LIN {X 0,Y 420.936,Z 312.19,A -85,B 0,C 180,E1 -10145.593,E2 -10145.593} C_VEL
LIN {X 0,Y 420.608,Z 319.802,A -85,B 0,C 180,E1 -10147.066,E2 -10147.066} C_VEL
LIN {X 0,Y 419.67,Z 336.36,A -85,B 0,C 180,E1 -10150.229,E2 -10150.229} C_VEL
LIN {X 0,Y 419.347,Z 341.705,A -85,B 0,C 180,E1 -10151.243,E2 -10151.243} C_VEL
LIN {X 0,Y 423.117,Z 368.844,A -85,B 0,C 180,E1 -10151.869,E2 -10151.869} C_VEL
LIN {X 0,Y 422.215,Z 450.861,A -85,B 0,C 180,E1 -10153.283,E2 -10153.283} C_VEL
LIN {X 0,Y 421.716,Z 464.725,A -85,B 0,C 180,E1 -10153.73,E2 -10153.73} C_VEL
LIN {X 0,Y 421.153,Z 477.157,A -85,B 0,C 180,E1 -10154.329,E2 -10154.329} C_VEL
LIN {X 0,Y 420.469,Z 489.063,A -85,B 0,C 180,E1 -10155.109,E2 -10155.109} C_VEL
LIN {X 0,Y 419.724,Z 501.027,A -85,B 0,C 180,E1 -10156.121,E2 -10156.121} C_VEL
LIN {X 0,Y 419.11,Z 510.84,A -85,B 0,C 180,E1 -10157.163,E2 -10157.163} C_VEL
LIN {X 0,Y 418.517,Z 520.102,A -85,B 0,C 180,E1 -10158.375,E2 -10158.375} C_VEL
LIN {X 0,Y 417.911,Z 529.108,A -85,B 0,C 180,E1 -10159.83,E2 -10159.83} C_VEL
LIN {X 0,Y 417.535,Z 536.352,A -85,B 0,C 180,E1 -10161.287,E2 -10161.287} C_VEL
LIN {X 0,Y 417.265,Z 542.12,A -85,B 0,C 180,E1 -10162.743,E2 -10162.743} C_VEL
LIN {X 0,Y 417.096,Z 546.655,A -85,B 0,C 180,E1 -10164.198,E2 -10164.198} C_VEL
LIN {X 0,Y 417.128,Z 549.047,A -85,B 0,C 180,E1 -10165.168,E2 -10165.168} C_VEL
LIN {X 0,Y 417.017,Z 550.997,A -85,B 0,C 180,E1 -10166.135,E2 -10166.135} C_VEL
LIN {X 0,Y 417.061,Z 552.532,A -85,B 0,C 180,E1 -10167.103,E2 -10167.103} C_VEL
LIN {X 0,Y 417.072,Z 553.609,A -85,B 0,C 180,E1 -10168.069,E2 -10168.069} C_VEL
LIN {X 0,Y 417.027,Z 554.572,A -85,B 0,C 180,E1 -10170.001,E2 -10170.001} C_VEL
LIN {X 0,Y 417.013,Z 554.471,A -85,B 0,C 180,E1 -10170.966,E2 -10170.966} C_VEL
LIN {X 0,Y 417.069,Z 553.941,A -85,B 0,C 180,E1 -10171.932,E2 -10171.932} C_VEL
LIN {X 0,Y 417.015,Z 551.682,A -85,B 0,C 180,E1 -10173.866,E2 -10173.866} C_VEL
LIN {X 0,Y 417.122,Z 548.885,A -85,B 0,C 180,E1 -10175.318,E2 -10175.318} C_VEL
LIN {X 0,Y 417.233,Z 545.071,A -85,B 0,C 180,E1 -10176.772,E2 -10176.772} C_VEL
LIN {X 0,Y 417.462,Z 540.144,A -85,B 0,C 180,E1 -10178.228,E2 -10178.228} C_VEL
LIN {X 0,Y 417.839,Z 533.958,A -85,B 0,C 180,E1 -10179.683,E2 -10179.683} C_VEL
LIN {X 0,Y 418.415,Z 526.279,A -85,B 0,C 180,E1 -10181.138,E2 -10181.138} C_VEL
LIN {X 0,Y 419.256,Z 516.655,A -85,B 0,C 180,E1 -10182.587,E2 -10182.587} C_VEL
LIN {X 0,Y 419.98,Z 506.28,A -85,B 0,C 180,E1 -10183.85,E2 -10183.85} C_VEL
LIN {X 0,Y 420.831,Z 495.628,A -85,B 0,C 180,E1 -10184.879,E2 -10184.879} C_VEL
LIN {X 0,Y 421.61,Z 484.753,A -85,B 0,C 180,E1 -10185.717,E2 -10185.717} C_VEL
LIN {X 0,Y 422.418,Z 472.754,A -85,B 0,C 180,E1 -10186.43,E2 -10186.43} C_VEL
LIN {X 0,Y 423.072,Z 459.606,A -85,B 0,C 180,E1 -10186.994,E2 -10186.994} C_VEL
LIN {X 0,Y 423.504,Z 446.445,A -85,B 0,C 180,E1 -10187.349,E2 -10187.349} C_VEL
LIN {X 0,Y 424.419,Z 367.986,A -85,B 0,C 180,E1 -10188.705,E2 -10188.705} C_VEL
LIN {X 0,Y 421.072,Z 347.455,A -85,B 0,C 180,E1 -10189.25,E2 -10189.25} C_VEL
LIN {X 0,Y 419.953,Z 341.257,A -85,B 0,C 180,E1 -10189.452,E2 -10189.452} C_VEL
LIN {X 0,Y 421.087,Z 324.061,A -85,B 0,C 180,E1 -10192.794,E2 -10192.794} C_VEL
LIN {X 0,Y 421.677,Z 314.787,A -85,B 0,C 180,E1 -10194.625,E2 -10194.625} C_VEL
LIN {X 0,Y 419.681,Z 304.414,A -85,B 0,C 180,E1 -10196.881,E2 -10196.881} C_VEL
LIN {X 0,Y 418.324,Z 298.383,A -85,B 0,C 180,E1 -10198.266,E2 -10198.266} C_VEL
LIN {X 0,Y 418.214,Z 298.393,A -85,B 0,C 180,E1 -10201.396,E2 -10201.396} C_VEL
LIN {X 0,Y 418.267,Z 298.386,A -85,B 0,C 180,E1 -10204.58,E2 -10204.58} C_VEL
LIN {X 0,Y 418.228,Z 298.389,A -85,B 0,C 180,E1 -10207.833,E2 -10207.833} C_VEL
LIN {X 0,Y 418.223,Z 298.389,A -85,B 0,C 180,E1 -10210.948,E2 -10210.948} C_VEL
LIN {X 0,Y 418.21,Z 298.389,A -85,B 0,C 180,E1 -10213.729,E2 -10213.729} C_VEL
LIN {X 0,Y 418.21,Z 298.393,A -85,B 0,C 180,E1 -10216.448,E2 -10216.448} C_VEL
LIN {X 0,Y 418.223,Z 298.386,A -85,B 0,C 180,E1 -10219.13,E2 -10219.13} C_VEL
LIN {X 0,Y 418.227,Z 298.386,A -85,B 0,C 180,E1 -10222.167,E2 -10222.167} C_VEL
LIN {X 0,Y 418.265,Z 298.378,A -85,B 0,C 180,E1 -10225.42,E2 -10225.42} C_VEL
LIN {X 0,Y 418.211,Z 298.39,A -85,B 0,C 180,E1 -10228.604,E2 -10228.604} C_VEL
LIN {X 0,Y 418.291,Z 298.377,A -85,B 0,C 180,E1 -10231.936,E2 -10231.936} C_VEL
LIN {X 0,Y 418.29,Z 298.383,A -85,B 0,C 180,E1 -10235.162,E2 -10235.162} C_VEL
LIN {X 0,Y 418.233,Z 298.383,A -85,B 0,C 180,E1 -10238.303,E2 -10238.303} C_VEL
LIN {X 0,Y 418.283,Z 298.379,A -85,B 0,C 180,E1 -10241.383,E2 -10241.383} C_VEL
LIN {X 0,Y 418.302,Z 298.373,A -85,B 0,C 180,E1 -10244.406,E2 -10244.406} C_VEL
LIN {X 0,Y 418.354,Z 298.37,A -85,B 0,C 180,E1 -10247.385,E2 -10247.385} C_VEL
LIN {X 0,Y 418.34,Z 298.367,A -85,B 0,C 180,E1 -10250.328,E2 -10250.328} C_VEL
LIN {X 0,Y 418.491,Z 298.351,A -85,B 0,C 180,E1 -10253.249,E2 -10253.249} C_VEL
LIN {X 0,Y 418.338,Z 298.365,A -85,B 0,C 180,E1 -10255.181,E2 -10255.181} C_VEL
LIN {X 0,Y 418.541,Z 298.343,A -85,B 0,C 180,E1 -10258.075,E2 -10258.075} C_VEL
LIN {X 0,Y 418.669,Z 298.329,A -85,B 0,C 180,E1 -10260,E2 -10260} C_VEL
LIN {X 0,Y 418.5,Z 298.344,A -85,B 0,C 180,E1 -10262.888,E2 -10262.888} C_VEL
LIN {X 0,Y 418.489,Z 298.349,A -85,B 0,C 180,E1 -10266.751,E2 -10266.751} C_VEL
LIN {X 0,Y 418.399,Z 298.364,A -85,B 0,C 180,E1 -10268.695,E2 -10268.695} C_VEL
LIN {X 0,Y 418.313,Z 298.372,A -85,B 0,C 180,E1 -10271.631,E2 -10271.631} C_VEL
LIN {X 0,Y 418.302,Z 298.381,A -85,B 0,C 180,E1 -10274.597,E2 -10274.597} C_VEL
LIN {X 0,Y 418.287,Z 298.376,A -85,B 0,C 180,E1 -10277.604,E2 -10277.604} C_VEL
LIN {X 0,Y 418.249,Z 298.384,A -85,B 0,C 180,E1 -10280.663,E2 -10280.663} C_VEL
LIN {X 0,Y 418.276,Z 298.377,A -85,B 0,C 180,E1 -10283.782,E2 -10283.782} C_VEL
LIN {X 0,Y 418.309,Z 298.376,A -85,B 0,C 180,E1 -10287.07,E2 -10287.07} C_VEL
LIN {X 0,Y 418.243,Z 298.382,A -85,B 0,C 180,E1 -10290.272,E2 -10290.272} C_VEL
LIN {X 0,Y 418.247,Z 298.382,A -85,B 0,C 180,E1 -10293.677,E2 -10293.677} C_VEL
LIN {X 0,Y 418.239,Z 298.386,A -85,B 0,C 180,E1 -10297.224,E2 -10297.224} C_VEL
LIN {X 0,Y 418.246,Z 298.383,A -85,B 0,C 180,E1 -10299.683,E2 -10299.683} C_VEL
LIN {X 0,Y 418.229,Z 298.385,A -85,B 0,C 180,E1 -10302.321,E2 -10302.321} C_VEL
LIN {X 0,Y 418.235,Z 298.387,A -85,B 0,C 180,E1 -10305.109,E2 -10305.109} C_VEL
LIN {X 0,Y 418.239,Z 298.388,A -85,B 0,C 180,E1 -10307.767,E2 -10307.767} C_VEL
LIN {X 0,Y 418.245,Z 298.386,A -85,B 0,C 180,E1 -10310.621,E2 -10310.621} C_VEL
LIN {X 0,Y 418.243,Z 298.386,A -85,B 0,C 180,E1 -10313.976,E2 -10313.976} C_VEL
LIN {X 0,Y 418.242,Z 298.389,A -85,B 0,C 180,E1 -10317.302,E2 -10317.302} C_VEL
LIN {X 0,Y 420.231,Z 307.957,A -85,B 0,C 180,E1 -10319.608,E2 -10319.608} C_VEL
LIN {X 0,Y 420.352,Z 312.594,A -85,B 0,C 180,E1 -10320.628,E2 -10320.628} C_VEL
LIN {X 0,Y 424.73,Z 331.843,A -85,B 0,C 180,E1 -10321.226,E2 -10321.226} C_VEL
LIN {X 0,Y 424.235,Z 375.558,A -85,B 0,C 180,E1 -10321.98,E2 -10321.98} C_VEL
LIN {X 0,Y 423.578,Z 420.934,A -85,B 0,C 180,E1 -10322.786,E2 -10322.786} C_VEL
LIN {X 0,Y 423.113,Z 434.256,A -85,B 0,C 180,E1 -10323.221,E2 -10323.221} C_VEL
LIN {X 0,Y 422.72,Z 446.148,A -85,B 0,C 180,E1 -10323.801,E2 -10323.801} C_VEL
LIN {X 0,Y 422.119,Z 456.766,A -85,B 0,C 180,E1 -10324.481,E2 -10324.481} C_VEL
LIN {X 0,Y 421.392,Z 467.515,A -85,B 0,C 180,E1 -10325.358,E2 -10325.358} C_VEL
LIN {X 0,Y 420.636,Z 477.399,A -85,B 0,C 180,E1 -10326.36,E2 -10326.36} C_VEL
LIN {X 0,Y 419.834,Z 487.413,A -85,B 0,C 180,E1 -10327.614,E2 -10327.614} C_VEL
LIN {X 0,Y 419.135,Z 495.554,A -85,B 0,C 180,E1 -10328.868,E2 -10328.868} C_VEL
LIN {X 0,Y 418.624,Z 502.01,A -85,B 0,C 180,E1 -10330.076,E2 -10330.076} C_VEL
LIN {X 0,Y 418.073,Z 507.767,A -85,B 0,C 180,E1 -10331.373,E2 -10331.373} C_VEL
LIN {X 0,Y 417.697,Z 513.126,A -85,B 0,C 180,E1 -10332.875,E2 -10332.875} C_VEL
LIN {X 0,Y 417.411,Z 517.248,A -85,B 0,C 180,E1 -10334.372,E2 -10334.372} C_VEL
LIN {X 0,Y 417.232,Z 519.362,A -85,B 0,C 180,E1 -10335.364,E2 -10335.364} C_VEL
LIN {X 0,Y 417.1,Z 521.024,A -85,B 0,C 180,E1 -10336.355,E2 -10336.355} C_VEL
LIN {X 0,Y 417.067,Z 522.941,A -85,B 0,C 180,E1 -10338.141,E2 -10338.141} C_VEL
LIN {X 0,Y 416.992,Z 523.472,A -85,B 0,C 180,E1 -10339.316,E2 -10339.316} C_VEL
LIN {X 0,Y 416.972,Z 523.075,A -85,B 0,C 180,E1 -10341.275,E2 -10341.275} C_VEL
LIN {X 0,Y 417.042,Z 522.162,A -85,B 0,C 180,E1 -10342.329,E2 -10342.329} C_VEL
LIN {X 0,Y 416.402,Z 521.209,A -85,B 0,C 180,E1 -10343.123,E2 -10343.123} C_VEL
LIN {X 0,Y 413.577,Z 519.17,A -85,B 0,C 180,E1 -10344.407,E2 -10344.407} C_VEL
LIN {X 0,Y 411.247,Z 517.028,A -85,B 0,C 180,E1 -10345.427,E2 -10345.427} C_VEL
LIN {X 0,Y 410.348,Z 515.063,A -85,B 0,C 180,E1 -10346.2,E2 -10346.2} C_VEL
LIN {X 0,Y 410.33,Z 514.318,A -85,B 0,C 180,E1 -10346.457,E2 -10346.457} C_VEL
LIN {X 0,Y 410.597,Z 509.016,A -85,B 0,C 180,E1 -10348.038,E2 -10348.038} C_VEL
LIN {X 0,Y 411.028,Z 502.734,A -85,B 0,C 180,E1 -10349.51,E2 -10349.51} C_VEL
LIN {X 0,Y 411.621,Z 494.875,A -85,B 0,C 180,E1 -10350.978,E2 -10350.978} C_VEL
LIN {X 0,Y 412.2,Z 485.137,A -85,B 0,C 180,E1 -10352.442,E2 -10352.442} C_VEL
LIN {X 0,Y 412.852,Z 474.969,A -85,B 0,C 180,E1 -10353.659,E2 -10353.659} C_VEL
LIN {X 0,Y 413.737,Z 464.843,A -85,B 0,C 180,E1 -10354.627,E2 -10354.627} C_VEL
LIN {X 0,Y 414.35,Z 453.869,A -85,B 0,C 180,E1 -10355.474,E2 -10355.474} C_VEL
LIN {X 0,Y 414.886,Z 441.713,A -85,B 0,C 180,E1 -10356.199,E2 -10356.199} C_VEL
LIN {X 0,Y 415.155,Z 428.961,A -85,B 0,C 180,E1 -10356.744,E2 -10356.744} C_VEL
LIN {X 0,Y 415.591,Z 416.702,A -85,B 0,C 180,E1 -10357.072,E2 -10357.072} C_VEL
LIN {X 0,Y 416.521,Z 332.666,A -85,B 0,C 180,E1 -10358.526,E2 -10358.526} C_VEL
LIN {X 0,Y 412.813,Z 312.758,A -85,B 0,C 180,E1 -10359.034,E2 -10359.034} C_VEL
LIN {X 0,Y 412.829,Z 308.131,A -85,B 0,C 180,E1 -10360.049,E2 -10360.049} C_VEL
LIN {X 0,Y 411.363,Z 299.247,A -85,B 0,C 180,E1 -10362.142,E2 -10362.142} C_VEL
LIN {X 0,Y 411.246,Z 299.256,A -85,B 0,C 180,E1 -10365.868,E2 -10365.868} C_VEL
LIN {X 0,Y 411.216,Z 299.259,A -85,B 0,C 180,E1 -10368.948,E2 -10368.948} C_VEL
LIN {X 0,Y 411.197,Z 299.266,A -85,B 0,C 180,E1 -10372.64,E2 -10372.64} C_VEL
LIN {X 0,Y 411.179,Z 299.263,A -85,B 0,C 180,E1 -10375.296,E2 -10375.296} C_VEL
LIN {X 0,Y 411.173,Z 299.27,A -85,B 0,C 180,E1 -10378.592,E2 -10378.592} C_VEL
LIN {X 0,Y 411.161,Z 299.265,A -85,B 0,C 180,E1 -10381.997,E2 -10381.997} C_VEL
LIN {X 0,Y 411.205,Z 299.266,A -85,B 0,C 180,E1 -10384.877,E2 -10384.877} C_VEL
LIN {X 0,Y 411.192,Z 299.261,A -85,B 0,C 180,E1 -10388.166,E2 -10388.166} C_VEL
LIN {X 0,Y 411.158,Z 299.265,A -85,B 0,C 180,E1 -10391.806,E2 -10391.806} C_VEL
LIN {X 0,Y 411.17,Z 299.266,A -85,B 0,C 180,E1 -10395.509,E2 -10395.509} C_VEL
LIN {X 0,Y 411.151,Z 299.268,A -85,B 0,C 180,E1 -10398.772,E2 -10398.772} C_VEL
LIN {X 0,Y 411.182,Z 299.262,A -85,B 0,C 180,E1 -10402.025,E2 -10402.025} C_VEL
LIN {X 0,Y 411.198,Z 299.264,A -85,B 0,C 180,E1 -10405.666,E2 -10405.666} C_VEL
LIN {X 0,Y 411.182,Z 299.265,A -85,B 0,C 180,E1 -10409.152,E2 -10409.152} C_VEL
LIN {X 0,Y 411.251,Z 299.253,A -85,B 0,C 180,E1 -10412.522,E2 -10412.522} C_VEL
LIN {X 0,Y 411.204,Z 299.265,A -85,B 0,C 180,E1 -10415.783,E2 -10415.783} C_VEL
LIN {X 0,Y 411.188,Z 299.261,A -85,B 0,C 180,E1 -10418.966,E2 -10418.966} C_VEL
LIN {X 0,Y 411.245,Z 299.258,A -85,B 0,C 180,E1 -10422.085,E2 -10422.085} C_VEL
LIN {X 0,Y 411.255,Z 299.253,A -85,B 0,C 180,E1 -10425.147,E2 -10425.147} C_VEL
LIN {X 0,Y 411.275,Z 299.256,A -85,B 0,C 180,E1 -10428.167,E2 -10428.167} C_VEL
LIN {X 0,Y 411.343,Z 299.242,A -85,B 0,C 180,E1 -10431.155,E2 -10431.155} C_VEL
LIN {X 0,Y 411.45,Z 299.236,A -85,B 0,C 180,E1 -10434.118,E2 -10434.118} C_VEL
LIN {X 0,Y 411.503,Z 299.227,A -85,B 0,C 180,E1 -10438.043,E2 -10438.043} C_VEL
LIN {X 0,Y 411.631,Z 299.21,A -85,B 0,C 180,E1 -10440,E2 -10440} C_VEL
LIN {X 0,Y 411.449,Z 299.23,A -85,B 0,C 180,E1 -10442.937,E2 -10442.937} C_VEL
LIN {X 0,Y 411.448,Z 299.232,A -85,B 0,C 180,E1 -10446.867,E2 -10446.867} C_VEL
LIN {X 0,Y 411.286,Z 299.249,A -85,B 0,C 180,E1 -10449.839,E2 -10449.839} C_VEL
LIN {X 0,Y 411.297,Z 299.25,A -85,B 0,C 180,E1 -10453.105,E2 -10453.105} C_VEL
LIN {X 0,Y 411.255,Z 299.259,A -85,B 0,C 180,E1 -10456.869,E2 -10456.869} C_VEL
LIN {X 0,Y 411.223,Z 299.257,A -85,B 0,C 180,E1 -10459.987,E2 -10459.987} C_VEL
LIN {X 0,Y 411.196,Z 299.265,A -85,B 0,C 180,E1 -10463.148,E2 -10463.148} C_VEL
LIN {X 0,Y 411.231,Z 299.257,A -85,B 0,C 180,E1 -10466.382,E2 -10466.382} C_VEL
LIN {X 0,Y 411.206,Z 299.26,A -85,B 0,C 180,E1 -10469.712,E2 -10469.712} C_VEL
LIN {X 0,Y 411.201,Z 299.267,A -85,B 0,C 180,E1 -10473.157,E2 -10473.157} C_VEL
LIN {X 0,Y 411.19,Z 299.261,A -85,B 0,C 180,E1 -10476.554,E2 -10476.554} C_VEL
LIN {X 0,Y 411.214,Z 299.261,A -85,B 0,C 180,E1 -10479.73,E2 -10479.73} C_VEL
LIN {X 0,Y 411.174,Z 299.266,A -85,B 0,C 180,E1 -10483.134,E2 -10483.134} C_VEL
LIN {X 0,Y 411.164,Z 299.267,A -85,B 0,C 180,E1 -10485.882,E2 -10485.882} C_VEL
LIN {X 0,Y 411.16,Z 299.265,A -85,B 0,C 180,E1 -10488.773,E2 -10488.773} C_VEL
LIN {X 0,Y 411.189,Z 299.265,A -85,B 0,C 180,E1 -10492.027,E2 -10492.027} C_VEL
LIN {X 0,Y 411.204,Z 299.265,A -85,B 0,C 180,E1 -10495.667,E2 -10495.667} C_VEL
LIN {X 0,Y 411.188,Z 299.261,A -85,B 0,C 180,E1 -10499.153,E2 -10499.153} C_VEL
LIN {X 0,Y 411.314,Z 299.353,A -85,B 0,C 180,E1 -10502.527,E2 -10502.527} C_VEL
LIN {X 0,Y 413.911,Z 312.994,A -85,B 0,C 180,E1 -10505.419,E2 -10505.419} C_VEL
LIN {X 0,Y 413.761,Z 319.175,A -85,B 0,C 180,E1 -10506.642,E2 -10506.642} C_VEL
LIN {X 0,Y 412.683,Z 336.91,A -85,B 0,C 180,E1 -10510.087,E2 -10510.087} C_VEL
LIN {X 0,Y 412.408,Z 341.367,A -85,B 0,C 180,E1 -10510.947,E2 -10510.947} C_VEL
LIN {X 0,Y 416.297,Z 369.883,A -85,B 0,C 180,E1 -10511.629,E2 -10511.629} C_VEL
LIN {X 0,Y 415.357,Z 450.171,A -85,B 0,C 180,E1 -10513.03,E2 -10513.03} C_VEL
LIN {X 0,Y 414.873,Z 463.413,A -85,B 0,C 180,E1 -10513.454,E2 -10513.454} C_VEL
LIN {X 0,Y 414.312,Z 476.161,A -85,B 0,C 180,E1 -10514.063,E2 -10514.063} C_VEL
LIN {X 0,Y 413.544,Z 488.258,A -85,B 0,C 180,E1 -10514.854,E2 -10514.854} C_VEL
LIN {X 0,Y 412.829,Z 499.823,A -85,B 0,C 180,E1 -10515.836,E2 -10515.836} C_VEL
LIN {X 0,Y 412.16,Z 510.297,A -85,B 0,C 180,E1 -10516.951,E2 -10516.951} C_VEL
LIN {X 0,Y 411.528,Z 519.568,A -85,B 0,C 180,E1 -10518.175,E2 -10518.175} C_VEL
LIN {X 0,Y 410.87,Z 528.62,A -85,B 0,C 180,E1 -10519.654,E2 -10519.654} C_VEL
LIN {X 0,Y 410.479,Z 535.909,A -85,B 0,C 180,E1 -10521.136,E2 -10521.136} C_VEL
LIN {X 0,Y 410.183,Z 541.721,A -85,B 0,C 180,E1 -10522.618,E2 -10522.618} C_VEL
LIN {X 0,Y 410.001,Z 546.289,A -85,B 0,C 180,E1 -10524.097,E2 -10524.097} C_VEL
LIN {X 0,Y 410.034,Z 548.697,A -85,B 0,C 180,E1 -10525.084,E2 -10525.084} C_VEL
LIN {X 0,Y 409.936,Z 550.662,A -85,B 0,C 180,E1 -10526.068,E2 -10526.068} C_VEL
LIN {X 0,Y 409.959,Z 552.214,A -85,B 0,C 180,E1 -10527.053,E2 -10527.053} C_VEL
LIN {X 0,Y 410,Z 553.313,A -85,B 0,C 180,E1 -10528.036,E2 -10528.036} C_VEL
LIN {X 0,Y 409.948,Z 554.301,A -85,B 0,C 180,E1 -10530.001,E2 -10530.001} C_VEL
LIN {X 0,Y 409.938,Z 554.216,A -85,B 0,C 180,E1 -10530.983,E2 -10530.983} C_VEL
LIN {X 0,Y 409.997,Z 553.708,A -85,B 0,C 180,E1 -10531.965,E2 -10531.965} C_VEL
LIN {X 0,Y 409.933,Z 551.474,A -85,B 0,C 180,E1 -10533.933,E2 -10533.933} C_VEL
LIN {X 0,Y 410.018,Z 548.704,A -85,B 0,C 180,E1 -10535.41,E2 -10535.41} C_VEL
LIN {X 0,Y 410.165,Z 544.919,A -85,B 0,C 180,E1 -10536.889,E2 -10536.889} C_VEL
LIN {X 0,Y 410.417,Z 540.024,A -85,B 0,C 180,E1 -10538.37,E2 -10538.37} C_VEL
LIN {X 0,Y 410.817,Z 533.875,A -85,B 0,C 180,E1 -10539.851,E2 -10539.851} C_VEL
LIN {X 0,Y 411.435,Z 526.251,A -85,B 0,C 180,E1 -10541.329,E2 -10541.329} C_VEL
LIN {X 0,Y 412.157,Z 518.468,A -85,B 0,C 180,E1 -10542.557,E2 -10542.557} C_VEL
LIN {X 0,Y 412.902,Z 508.984,A -85,B 0,C 180,E1 -10543.786,E2 -10543.786} C_VEL
LIN {X 0,Y 413.735,Z 498.496,A -85,B 0,C 180,E1 -10544.888,E2 -10544.888} C_VEL
LIN {X 0,Y 414.68,Z 486.836,A -85,B 0,C 180,E1 -10545.86,E2 -10545.86} C_VEL
LIN {X 0,Y 415.581,Z 474.397,A -85,B 0,C 180,E1 -10546.645,E2 -10546.645} C_VEL
LIN {X 0,Y 416.266,Z 461.319,A -85,B 0,C 180,E1 -10547.249,E2 -10547.249} C_VEL
LIN {X 0,Y 416.812,Z 448.275,A -85,B 0,C 180,E1 -10547.637,E2 -10547.637} C_VEL
LIN {X 0,Y 417.763,Z 368.347,A -85,B 0,C 180,E1 -10549.049,E2 -10549.049} C_VEL
LIN {X 0,Y 413.85,Z 345.109,A -85,B 0,C 180,E1 -10549.689,E2 -10549.689} C_VEL
LIN {X 0,Y 413.093,Z 341.048,A -85,B 0,C 180,E1 -10549.824,E2 -10549.824} C_VEL
LIN {X 0,Y 414.215,Z 325.143,A -85,B 0,C 180,E1 -10552.97,E2 -10552.97} C_VEL
LIN {X 0,Y 414.792,Z 317.366,A -85,B 0,C 180,E1 -10554.527,E2 -10554.527} C_VEL
LIN {X 0,Y 413.883,Z 311.29,A -85,B 0,C 180,E1 -10555.845,E2 -10555.845} C_VEL
LIN {X 0,Y 411.268,Z 299.263,A -85,B 0,C 180,E1 -10558.586,E2 -10558.586} C_VEL
LIN {X 0,Y 411.168,Z 299.273,A -85,B 0,C 180,E1 -10561.997,E2 -10561.997} C_VEL
LIN {X 0,Y 411.213,Z 299.262,A -85,B 0,C 180,E1 -10564.878,E2 -10564.878} C_VEL
LIN {X 0,Y 411.203,Z 299.265,A -85,B 0,C 180,E1 -10568.168,E2 -10568.168} C_VEL
LIN {X 0,Y 411.164,Z 299.267,A -85,B 0,C 180,E1 -10571.228,E2 -10571.228} C_VEL
LIN {X 0,Y 411.177,Z 299.268,A -85,B 0,C 180,E1 -10574.49,E2 -10574.49} C_VEL
LIN {X 0,Y 411.178,Z 299.265,A -85,B 0,C 180,E1 -10578.194,E2 -10578.194} C_VEL
LIN {X 0,Y 411.215,Z 299.263,A -85,B 0,C 180,E1 -10580.775,E2 -10580.775} C_VEL
LIN {X 0,Y 411.198,Z 299.263,A -85,B 0,C 180,E1 -10584.471,E2 -10584.471} C_VEL
LIN {X 0,Y 411.207,Z 299.261,A -85,B 0,C 180,E1 -10586.873,E2 -10586.873} C_VEL
LIN {X 0,Y 411.233,Z 299.256,A -85,B 0,C 180,E1 -10590.644,E2 -10590.644} C_VEL
LIN {X 0,Y 411.237,Z 299.257,A -85,B 0,C 180,E1 -10593.619,E2 -10593.619} C_VEL
LIN {X 0,Y 411.202,Z 299.262,A -85,B 0,C 180,E1 -10596.852,E2 -10596.852} C_VEL
LIN {X 0,Y 411.214,Z 299.258,A -85,B 0,C 180,E1 -10600.05,E2 -10600.05} C_VEL
LIN {X 0,Y 411.262,Z 299.254,A -85,B 0,C 180,E1 -10603.131,E2 -10603.131} C_VEL
LIN {X 0,Y 411.305,Z 299.244,A -85,B 0,C 180,E1 -10606.896,E2 -10606.896} C_VEL
LIN {X 0,Y 411.292,Z 299.246,A -85,B 0,C 180,E1 -10610.161,E2 -10610.161} C_VEL
LIN {X 0,Y 411.455,Z 299.226,A -85,B 0,C 180,E1 -10613.133,E2 -10613.133} C_VEL
LIN {X 0,Y 411.309,Z 299.24,A -85,B 0,C 180,E1 -10615.099,E2 -10615.099} C_VEL
LIN {X 0,Y 411.51,Z 299.219,A -85,B 0,C 180,E1 -10618.042,E2 -10618.042} C_VEL
LIN {X 0,Y 411.638,Z 299.204,A -85,B 0,C 180,E1 -10620,E2 -10620} C_VEL
LIN {X 0,Y 411.456,Z 299.221,A -85,B 0,C 180,E1 -10622.937,E2 -10622.937} C_VEL
LIN {X 0,Y 411.457,Z 299.224,A -85,B 0,C 180,E1 -10626.867,E2 -10626.867} C_VEL
LIN {X 0,Y 411.353,Z 299.241,A -85,B 0,C 180,E1 -10628.845,E2 -10628.845} C_VEL
LIN {X 0,Y 411.282,Z 299.249,A -85,B 0,C 180,E1 -10631.833,E2 -10631.833} C_VEL
LIN {X 0,Y 411.259,Z 299.255,A -85,B 0,C 180,E1 -10634.853,E2 -10634.853} C_VEL
LIN {X 0,Y 411.251,Z 299.254,A -85,B 0,C 180,E1 -10637.915,E2 -10637.915} C_VEL
LIN {X 0,Y 411.195,Z 299.263,A -85,B 0,C 180,E1 -10641.034,E2 -10641.034} C_VEL
LIN {X 0,Y 411.22,Z 299.258,A -85,B 0,C 180,E1 -10644.216,E2 -10644.216} C_VEL
LIN {X 0,Y 411.258,Z 299.25,A -85,B 0,C 180,E1 -10647.478,E2 -10647.478} C_VEL
LIN {X 0,Y 411.189,Z 299.265,A -85,B 0,C 180,E1 -10650.848,E2 -10650.848} C_VEL
LIN {X 0,Y 411.205,Z 299.258,A -85,B 0,C 180,E1 -10654.334,E2 -10654.334} C_VEL
LIN {X 0,Y 411.192,Z 299.261,A -85,B 0,C 180,E1 -10657.974,E2 -10657.974} C_VEL
LIN {X 0,Y 411.163,Z 299.27,A -85,B 0,C 180,E1 -10661.228,E2 -10661.228} C_VEL
LIN {X 0,Y 411.175,Z 299.264,A -85,B 0,C 180,E1 -10664.49,E2 -10664.49} C_VEL
LIN {X 0,Y 411.177,Z 299.265,A -85,B 0,C 180,E1 -10668.195,E2 -10668.195} C_VEL
LIN {X 0,Y 411.211,Z 299.262,A -85,B 0,C 180,E1 -10670.775,E2 -10670.775} C_VEL
LIN {X 0,Y 411.198,Z 299.261,A -85,B 0,C 180,E1 -10674.471,E2 -10674.471} C_VEL
LIN {X 0,Y 411.233,Z 299.389,A -85,B 0,C 180,E1 -10677.057,E2 -10677.057} C_VEL
LIN {X 0,Y 413.22,Z 308.79,A -85,B 0,C 180,E1 -10679.32,E2 -10679.32} C_VEL
LIN {X 0,Y 413.532,Z 312.859,A -85,B 0,C 180,E1 -10680.245,E2 -10680.245} C_VEL
LIN {X 0,Y 418.242,Z 333.489,A -85,B 0,C 180,E1 -10680.902,E2 -10680.902} C_VEL
LIN {X 0,Y 416.916,Z 420.997,A -85,B 0,C 180,E1 -10682.45,E2 -10682.45} C_VEL
LIN {X 0,Y 416.42,Z 434.381,A -85,B 0,C 180,E1 -10682.891,E2 -10682.891} C_VEL
LIN {X 0,Y 415.995,Z 446.833,A -85,B 0,C 180,E1 -10683.511,E2 -10683.511} C_VEL
LIN {X 0,Y 415.272,Z 458.615,A -85,B 0,C 180,E1 -10684.299,E2 -10684.299} C_VEL
LIN {X 0,Y 414.394,Z 470.373,A -85,B 0,C 180,E1 -10685.315,E2 -10685.315} C_VEL
LIN {X 0,Y 413.607,Z 480.137,A -85,B 0,C 180,E1 -10686.372,E2 -10686.372} C_VEL
LIN {X 0,Y 412.891,Z 488.541,A -85,B 0,C 180,E1 -10687.481,E2 -10687.481} C_VEL
LIN {X 0,Y 412.166,Z 496.511,A -85,B 0,C 180,E1 -10688.756,E2 -10688.756} C_VEL
LIN {X 0,Y 411.445,Z 504.231,A -85,B 0,C 180,E1 -10690.284,E2 -10690.284} C_VEL
LIN {X 0,Y 410.841,Z 511.303,A -85,B 0,C 180,E1 -10692.066,E2 -10692.066} C_VEL
LIN {X 0,Y 410.525,Z 515.604,A -85,B 0,C 180,E1 -10693.475,E2 -10693.475} C_VEL
LIN {X 0,Y 410.204,Z 519.386,A -85,B 0,C 180,E1 -10695.108,E2 -10695.108} C_VEL
LIN {X 0,Y 410.057,Z 521.094,A -85,B 0,C 180,E1 -10696.116,E2 -10696.116} C_VEL
LIN {X 0,Y 410.001,Z 522.933,A -85,B 0,C 180,E1 -10697.704,E2 -10697.704} C_VEL
LIN {X 0,Y 409.931,Z 523.716,A -85,B 0,C 180,E1 -10699.129,E2 -10699.129} C_VEL
LIN {X 0,Y 409.864,Z 523.406,A -85,B 0,C 180,E1 -10701.122,E2 -10701.122} C_VEL
LIN {X 0,Y 409.952,Z 522.397,A -85,B 0,C 180,E1 -10702.342,E2 -10702.342} C_VEL
LIN {X 0,Y 410.119,Z 519.889,A -85,B 0,C 180,E1 -10704.098,E2 -10704.098} C_VEL
LIN {X 0,Y 410.164,Z 516.71,A -85,B 0,C 180,E1 -10705.577,E2 -10705.577} C_VEL
LIN {X 0,Y 410.33,Z 514.318,A -85,B 0,C 180,E1 -10706.457,E2 -10706.457} C_VEL
LIN {X 0,Y 409.85,Z 512.038,A -85,B 0,C 180,E1 -10707.216,E2 -10707.216} C_VEL
LIN {X 0,Y 407.25,Z 507.932,A -85,B 0,C 180,E1 -10708.43,E2 -10708.43} C_VEL
LIN {X 0,Y 404.688,Z 503.127,A -85,B 0,C 180,E1 -10709.604,E2 -10709.604} C_VEL
LIN {X 0,Y 404.272,Z 499.747,A -85,B 0,C 180,E1 -10710.29,E2 -10710.29} C_VEL
LIN {X 0,Y 404.875,Z 491.372,A -85,B 0,C 180,E1 -10711.74,E2 -10711.74} C_VEL
LIN {X 0,Y 405.413,Z 482.595,A -85,B 0,C 180,E1 -10712.981,E2 -10712.981} C_VEL
LIN {X 0,Y 406.122,Z 472.94,A -85,B 0,C 180,E1 -10714.093,E2 -10714.093} C_VEL
LIN {X 0,Y 407.028,Z 462.319,A -85,B 0,C 180,E1 -10715.076,E2 -10715.076} C_VEL
LIN {X 0,Y 407.609,Z 450.524,A -85,B 0,C 180,E1 -10715.937,E2 -10715.937} C_VEL
LIN {X 0,Y 408.126,Z 438.264,A -85,B 0,C 180,E1 -10716.612,E2 -10716.612} C_VEL
LIN {X 0,Y 408.432,Z 426.605,A -85,B 0,C 180,E1 -10717.073,E2 -10717.073} C_VEL
LIN {X 0,Y 408.777,Z 414.179,A -85,B 0,C 180,E1 -10717.377,E2 -10717.377} C_VEL
LIN {X 0,Y 409.674,Z 333.501,A -85,B 0,C 180,E1 -10718.788,E2 -10718.788} C_VEL
LIN {X 0,Y 405.881,Z 312.872,A -85,B 0,C 180,E1 -10719.351,E2 -10719.351} C_VEL
LIN {X 0,Y 405.823,Z 308.965,A -85,B 0,C 180,E1 -10720.224,E2 -10720.224} C_VEL
LIN {X 0,Y 404.304,Z 300.126,A -85,B 0,C 180,E1 -10722.326,E2 -10722.326} C_VEL
LIN {X 0,Y 404.215,Z 300.135,A -85,B 0,C 180,E1 -10726.151,E2 -10726.151} C_VEL
LIN {X 0,Y 404.16,Z 300.137,A -85,B 0,C 180,E1 -10729.292,E2 -10729.292} C_VEL
LIN {X 0,Y 404.144,Z 300.142,A -85,B 0,C 180,E1 -10732.83,E2 -10732.83} C_VEL
LIN {X 0,Y 404.131,Z 300.14,A -85,B 0,C 180,E1 -10735.769,E2 -10735.769} C_VEL
LIN {X 0,Y 404.151,Z 300.138,A -85,B 0,C 180,E1 -10739.602,E2 -10739.602} C_VEL
LIN {X 0,Y 404.137,Z 300.145,A -85,B 0,C 180,E1 -10742.621,E2 -10742.621} C_VEL
LIN {X 0,Y 404.176,Z 300.138,A -85,B 0,C 180,E1 -10745.189,E2 -10745.189} C_VEL
LIN {X 0,Y 404.132,Z 300.145,A -85,B 0,C 180,E1 -10748.758,E2 -10748.758} C_VEL
LIN {X 0,Y 404.104,Z 300.145,A -85,B 0,C 180,E1 -10751.597,E2 -10751.597} C_VEL
LIN {X 0,Y 404.138,Z 300.141,A -85,B 0,C 180,E1 -10754.521,E2 -10754.521} C_VEL
LIN {X 0,Y 404.126,Z 300.147,A -85,B 0,C 180,E1 -10757.294,E2 -10757.294} C_VEL
LIN {X 0,Y 404.128,Z 300.141,A -85,B 0,C 180,E1 -10759.95,E2 -10759.95} C_VEL
LIN {X 0,Y 404.128,Z 300.145,A -85,B 0,C 180,E1 -10763.125,E2 -10763.125} C_VEL
LIN {X 0,Y 404.138,Z 300.14,A -85,B 0,C 180,E1 -10766.187,E2 -10766.187} C_VEL
LIN {X 0,Y 404.138,Z 300.144,A -85,B 0,C 180,E1 -10769.714,E2 -10769.714} C_VEL
LIN {X 0,Y 404.185,Z 300.135,A -85,B 0,C 180,E1 -10773.122,E2 -10773.122} C_VEL
LIN {X 0,Y 404.162,Z 300.14,A -85,B 0,C 180,E1 -10775.333,E2 -10775.333} C_VEL
LIN {X 0,Y 404.13,Z 300.14,A -85,B 0,C 180,E1 -10778.58,E2 -10778.58} C_VEL
LIN {X 0,Y 404.202,Z 300.138,A -85,B 0,C 180,E1 -10781.762,E2 -10781.762} C_VEL
LIN {X 0,Y 404.202,Z 300.131,A -85,B 0,C 180,E1 -10784.882,E2 -10784.882} C_VEL
LIN {X 0,Y 404.247,Z 300.133,A -85,B 0,C 180,E1 -10787.958,E2 -10787.958} C_VEL
LIN {X 0,Y 404.28,Z 300.121,A -85,B 0,C 180,E1 -10790.999,E2 -10790.999} C_VEL
LIN {X 0,Y 404.397,Z 300.113,A -85,B 0,C 180,E1 -10794.015,E2 -10794.015} C_VEL
LIN {X 0,Y 404.472,Z 300.102,A -85,B 0,C 180,E1 -10798.009,E2 -10798.009} C_VEL
LIN {X 0,Y 404.6,Z 300.085,A -85,B 0,C 180,E1 -10800,E2 -10800} C_VEL
LIN {X 0,Y 404.408,Z 300.107,A -85,B 0,C 180,E1 -10802.989,E2 -10802.989} C_VEL
LIN {X 0,Y 404.414,Z 300.107,A -85,B 0,C 180,E1 -10805.985,E2 -10805.985} C_VEL
LIN {X 0,Y 404.283,Z 300.123,A -85,B 0,C 180,E1 -10809.001,E2 -10809.001} C_VEL
LIN {X 0,Y 404.249,Z 300.127,A -85,B 0,C 180,E1 -10812.042,E2 -10812.042} C_VEL
LIN {X 0,Y 404.199,Z 300.134,A -85,B 0,C 180,E1 -10815.118,E2 -10815.118} C_VEL
LIN {X 0,Y 404.203,Z 300.133,A -85,B 0,C 180,E1 -10818.239,E2 -10818.239} C_VEL
LIN {X 0,Y 404.131,Z 300.142,A -85,B 0,C 180,E1 -10821.42,E2 -10821.42} C_VEL
LIN {X 0,Y 404.17,Z 300.139,A -85,B 0,C 180,E1 -10824.666,E2 -10824.666} C_VEL
LIN {X 0,Y 404.192,Z 300.132,A -85,B 0,C 180,E1 -10828,E2 -10828} C_VEL
LIN {X 0,Y 404.142,Z 300.142,A -85,B 0,C 180,E1 -10831.561,E2 -10831.561} C_VEL
LIN {X 0,Y 404.18,Z 300.139,A -85,B 0,C 180,E1 -10835.017,E2 -10835.017} C_VEL
LIN {X 0,Y 404.154,Z 300.138,A -85,B 0,C 180,E1 -10838.757,E2 -10838.757} C_VEL
LIN {X 0,Y 404.12,Z 300.147,A -85,B 0,C 180,E1 -10841.601,E2 -10841.601} C_VEL
LIN {X 0,Y 404.145,Z 300.138,A -85,B 0,C 180,E1 -10844.524,E2 -10844.524} C_VEL
LIN {X 0,Y 404.133,Z 300.144,A -85,B 0,C 180,E1 -10847.297,E2 -10847.297} C_VEL
LIN {X 0,Y 404.166,Z 300.14,A -85,B 0,C 180,E1 -10849.956,E2 -10849.956} C_VEL
LIN {X 0,Y 404.133,Z 300.141,A -85,B 0,C 180,E1 -10853.126,E2 -10853.126} C_VEL
LIN {X 0,Y 404.143,Z 300.142,A -85,B 0,C 180,E1 -10856.189,E2 -10856.189} C_VEL
LIN {X 0,Y 404.144,Z 300.144,A -85,B 0,C 180,E1 -10859.716,E2 -10859.716} C_VEL
LIN {X 0,Y 404.278,Z 300.228,A -85,B 0,C 180,E1 -10862.312,E2 -10862.312} C_VEL
LIN {X 0,Y 406.839,Z 313.779,A -85,B 0,C 180,E1 -10865.235,E2 -10865.235} C_VEL
LIN {X 0,Y 406.908,Z 318.838,A -85,B 0,C 180,E1 -10866.263,E2 -10866.263} C_VEL
LIN {X 0,Y 405.668,Z 337.712,A -85,B 0,C 180,E1 -10869.992,E2 -10869.992} C_VEL
LIN {X 0,Y 405.445,Z 341.182,A -85,B 0,C 180,E1 -10870.673,E2 -10870.673} C_VEL
LIN {X 0,Y 409.453,Z 369.811,A -85,B 0,C 180,E1 -10871.36,E2 -10871.36} C_VEL
LIN {X 0,Y 408.512,Z 449.408,A -85,B 0,C 180,E1 -10872.77,E2 -10872.77} C_VEL
LIN {X 0,Y 408.018,Z 462.826,A -85,B 0,C 180,E1 -10873.2,E2 -10873.2} C_VEL
LIN {X 0,Y 407.461,Z 475.092,A -85,B 0,C 180,E1 -10873.788,E2 -10873.788} C_VEL
LIN {X 0,Y 406.656,Z 487.432,A -85,B 0,C 180,E1 -10874.591,E2 -10874.591} C_VEL
LIN {X 0,Y 405.907,Z 499.098,A -85,B 0,C 180,E1 -10875.589,E2 -10875.589} C_VEL
LIN {X 0,Y 405.192,Z 509.867,A -85,B 0,C 180,E1 -10876.746,E2 -10876.746} C_VEL
LIN {X 0,Y 404.553,Z 519.022,A -85,B 0,C 180,E1 -10877.968,E2 -10877.968} C_VEL
LIN {X 0,Y 403.823,Z 528.119,A -85,B 0,C 180,E1 -10879.471,E2 -10879.471} C_VEL
LIN {X 0,Y 403.4,Z 535.451,A -85,B 0,C 180,E1 -10880.98,E2 -10880.98} C_VEL
LIN {X 0,Y 403.129,Z 541.313,A -85,B 0,C 180,E1 -10882.488,E2 -10882.488} C_VEL
LIN {X 0,Y 402.938,Z 545.916,A -85,B 0,C 180,E1 -10883.994,E2 -10883.994} C_VEL
LIN {X 0,Y 402.942,Z 548.343,A -85,B 0,C 180,E1 -10884.998,E2 -10884.998} C_VEL
LIN {X 0,Y 402.857,Z 550.323,A -85,B 0,C 180,E1 -10885.999,E2 -10885.999} C_VEL
LIN {X 0,Y 402.859,Z 551.889,A -85,B 0,C 180,E1 -10887.001,E2 -10887.001} C_VEL
LIN {X 0,Y 402.912,Z 553.016,A -85,B 0,C 180,E1 -10888.001,E2 -10888.001} C_VEL
LIN {X 0,Y 402.871,Z 554.031,A -85,B 0,C 180,E1 -10890.001,E2 -10890.001} C_VEL
LIN {X 0,Y 402.866,Z 553.958,A -85,B 0,C 180,E1 -10891,E2 -10891} C_VEL
LIN {X 0,Y 402.907,Z 553.476,A -85,B 0,C 180,E1 -10892,E2 -10892} C_VEL
LIN {X 0,Y 402.853,Z 551.269,A -85,B 0,C 180,E1 -10894.002,E2 -10894.002} C_VEL
LIN {X 0,Y 402.916,Z 548.527,A -85,B 0,C 180,E1 -10895.506,E2 -10895.506} C_VEL
LIN {X 0,Y 403.078,Z 544.773,A -85,B 0,C 180,E1 -10897.011,E2 -10897.011} C_VEL
LIN {X 0,Y 403.359,Z 539.912,A -85,B 0,C 180,E1 -10898.517,E2 -10898.517} C_VEL
LIN {X 0,Y 403.809,Z 533.801,A -85,B 0,C 180,E1 -10900.023,E2 -10900.023} C_VEL
LIN {X 0,Y 404.437,Z 526.225,A -85,B 0,C 180,E1 -10901.528,E2 -10901.528} C_VEL
LIN {X 0,Y 405.213,Z 518.501,A -85,B 0,C 180,E1 -10902.776,E2 -10902.776} C_VEL
LIN {X 0,Y 405.982,Z 509.1,A -85,B 0,C 180,E1 -10904.026,E2 -10904.026} C_VEL
LIN {X 0,Y 406.887,Z 498.69,A -85,B 0,C 180,E1 -10905.144,E2 -10905.144} C_VEL
LIN {X 0,Y 407.88,Z 487.147,A -85,B 0,C 180,E1 -10906.132,E2 -10906.132} C_VEL
LIN {X 0,Y 408.826,Z 474.947,A -85,B 0,C 180,E1 -10906.928,E2 -10906.928} C_VEL
LIN {X 0,Y 409.567,Z 461.403,A -85,B 0,C 180,E1 -10907.572,E2 -10907.572} C_VEL
LIN {X 0,Y 410.147,Z 448.686,A -85,B 0,C 180,E1 -10907.965,E2 -10907.965} C_VEL
LIN {X 0,Y 411.145,Z 369.032,A -85,B 0,C 180,E1 -10909.399,E2 -10909.399} C_VEL
LIN {X 0,Y 407.397,Z 346.781,A -85,B 0,C 180,E1 -10910.028,E2 -10910.028} C_VEL
LIN {X 0,Y 406.242,Z 340.683,A -85,B 0,C 180,E1 -10910.243,E2 -10910.243} C_VEL
LIN {X 0,Y 407.512,Z 324.026,A -85,B 0,C 180,E1 -10913.6,E2 -10913.6} C_VEL
LIN {X 0,Y 407.834,Z 317.361,A -85,B 0,C 180,E1 -10914.974,E2 -10914.974} C_VEL
LIN {X 0,Y 405.521,Z 305.678,A -85,B 0,C 180,E1 -10917.628,E2 -10917.628} C_VEL
LIN {X 0,Y 404.199,Z 300.142,A -85,B 0,C 180,E1 -10918.991,E2 -10918.991} C_VEL
LIN {X 0,Y 404.143,Z 300.141,A -85,B 0,C 180,E1 -10922.622,E2 -10922.622} C_VEL
LIN {X 0,Y 404.183,Z 300.137,A -85,B 0,C 180,E1 -10925.19,E2 -10925.19} C_VEL
LIN {X 0,Y 404.152,Z 300.144,A -85,B 0,C 180,E1 -10928.757,E2 -10928.757} C_VEL
LIN {X 0,Y 404.124,Z 300.144,A -85,B 0,C 180,E1 -10931.599,E2 -10931.599} C_VEL
LIN {X 0,Y 404.146,Z 300.143,A -85,B 0,C 180,E1 -10934.522,E2 -10934.522} C_VEL
LIN {X 0,Y 404.137,Z 300.141,A -85,B 0,C 180,E1 -10937.295,E2 -10937.295} C_VEL
LIN {X 0,Y 404.17,Z 300.134,A -85,B 0,C 180,E1 -10939.955,E2 -10939.955} C_VEL
LIN {X 0,Y 404.136,Z 300.142,A -85,B 0,C 180,E1 -10943.125,E2 -10943.125} C_VEL
LIN {X 0,Y 404.145,Z 300.136,A -85,B 0,C 180,E1 -10946.187,E2 -10946.187} C_VEL
LIN {X 0,Y 404.145,Z 300.138,A -85,B 0,C 180,E1 -10949.715,E2 -10949.715} C_VEL
LIN {X 0,Y 404.195,Z 300.134,A -85,B 0,C 180,E1 -10953.123,E2 -10953.123} C_VEL
LIN {X 0,Y 404.177,Z 300.141,A -85,B 0,C 180,E1 -10955.334,E2 -10955.334} C_VEL
LIN {X 0,Y 404.138,Z 300.139,A -85,B 0,C 180,E1 -10958.58,E2 -10958.58} C_VEL
LIN {X 0,Y 404.21,Z 300.132,A -85,B 0,C 180,E1 -10961.762,E2 -10961.762} C_VEL
LIN {X 0,Y 404.206,Z 300.13,A -85,B 0,C 180,E1 -10964.882,E2 -10964.882} C_VEL
LIN {X 0,Y 404.255,Z 300.126,A -85,B 0,C 180,E1 -10967.958,E2 -10967.958} C_VEL
LIN {X 0,Y 404.404,Z 300.107,A -85,B 0,C 180,E1 -10972.129,E2 -10972.129} C_VEL
LIN {X 0,Y 404.421,Z 300.101,A -85,B 0,C 180,E1 -10974.015,E2 -10974.015} C_VEL
LIN {X 0,Y 404.479,Z 300.095,A -85,B 0,C 180,E1 -10978.008,E2 -10978.008} C_VEL
LIN {X 0,Y 404.608,Z 300.08,A -85,B 0,C 180,E1 -10980,E2 -10980} C_VEL
LIN {X 0,Y 404.415,Z 300.098,A -85,B 0,C 180,E1 -10982.988,E2 -10982.988} C_VEL
LIN {X 0,Y 404.408,Z 300.102,A -85,B 0,C 180,E1 -10986.987,E2 -10986.987} C_VEL
LIN {X 0,Y 404.257,Z 300.127,A -85,B 0,C 180,E1 -10990.012,E2 -10990.012} C_VEL
LIN {X 0,Y 404.265,Z 300.123,A -85,B 0,C 180,E1 -10993.211,E2 -10993.211} C_VEL
LIN {X 0,Y 404.215,Z 300.132,A -85,B 0,C 180,E1 -10997.007,E2 -10997.007} C_VEL
LIN {X 0,Y 404.163,Z 300.139,A -85,B 0,C 180,E1 -11000.352,E2 -11000.352} C_VEL
LIN {X 0,Y 404.163,Z 300.136,A -85,B 0,C 180,E1 -11003.575,E2 -11003.575} C_VEL
LIN {X 0,Y 404.183,Z 300.133,A -85,B 0,C 180,E1 -11005.766,E2 -11005.766} C_VEL
LIN {X 0,Y 404.194,Z 300.129,A -85,B 0,C 180,E1 -11008,E2 -11008} C_VEL
LIN {X 0,Y 404.138,Z 300.138,A -85,B 0,C 180,E1 -11011.558,E2 -11011.558} C_VEL
LIN {X 0,Y 404.184,Z 300.135,A -85,B 0,C 180,E1 -11015.016,E2 -11015.016} C_VEL
LIN {X 0,Y 404.152,Z 300.14,A -85,B 0,C 180,E1 -11018.757,E2 -11018.757} C_VEL
LIN {X 0,Y 404.123,Z 300.146,A -85,B 0,C 180,E1 -11021.6,E2 -11021.6} C_VEL
LIN {X 0,Y 404.145,Z 300.14,A -85,B 0,C 180,E1 -11024.522,E2 -11024.522} C_VEL
LIN {X 0,Y 404.136,Z 300.145,A -85,B 0,C 180,E1 -11027.296,E2 -11027.296} C_VEL
LIN {X 0,Y 404.169,Z 300.14,A -85,B 0,C 180,E1 -11029.955,E2 -11029.955} C_VEL
LIN {X 0,Y 404.136,Z 300.144,A -85,B 0,C 180,E1 -11033.125,E2 -11033.125} C_VEL
LIN {X 0,Y 404.149,Z 300.145,A -85,B 0,C 180,E1 -11036.188,E2 -11036.188} C_VEL
LIN {X 0,Y 404.19,Z 300.255,A -85,B 0,C 180,E1 -11036.716,E2 -11036.716} C_VEL
LIN {X 0,Y 406.433,Z 310.922,A -85,B 0,C 180,E1 -11039.329,E2 -11039.329} C_VEL
LIN {X 0,Y 406.741,Z 313.458,A -85,B 0,C 180,E1 -11039.864,E2 -11039.864} C_VEL
LIN {X 0,Y 411.321,Z 332.813,A -85,B 0,C 180,E1 -11040.498,E2 -11040.498} C_VEL
LIN {X 0,Y 411.652,Z 336.493,A -85,B 0,C 180,E1 -11040.586,E2 -11040.586} C_VEL
LIN {X 0,Y 410.276,Z 421.133,A -85,B 0,C 180,E1 -11042.104,E2 -11042.104} C_VEL
LIN {X 0,Y 409.752,Z 434.476,A -85,B 0,C 180,E1 -11042.548,E2 -11042.548} C_VEL
LIN {X 0,Y 409.278,Z 447.158,A -85,B 0,C 180,E1 -11043.187,E2 -11043.187} C_VEL
LIN {X 0,Y 408.543,Z 458.826,A -85,B 0,C 180,E1 -11043.981,E2 -11043.981} C_VEL
LIN {X 0,Y 407.62,Z 470.59,A -85,B 0,C 180,E1 -11045.012,E2 -11045.012} C_VEL
LIN {X 0,Y 406.713,Z 481.267,A -85,B 0,C 180,E1 -11046.198,E2 -11046.198} C_VEL
LIN {X 0,Y 405.723,Z 491.292,A -85,B 0,C 180,E1 -11047.599,E2 -11047.599} C_VEL
LIN {X 0,Y 405.055,Z 498.828,A -85,B 0,C 180,E1 -11048.898,E2 -11048.898} C_VEL
LIN {X 0,Y 404.355,Z 506.177,A -85,B 0,C 180,E1 -11050.453,E2 -11050.453} C_VEL
LIN {X 0,Y 403.859,Z 511.09,A -85,B 0,C 180,E1 -11051.745,E2 -11051.745} C_VEL
LIN {X 0,Y 403.502,Z 515.904,A -85,B 0,C 180,E1 -11053.328,E2 -11053.328} C_VEL
LIN {X 0,Y 403.179,Z 519.387,A -85,B 0,C 180,E1 -11054.842,E2 -11054.842} C_VEL
LIN {X 0,Y 402.996,Z 521.167,A -85,B 0,C 180,E1 -11055.868,E2 -11055.868} C_VEL
LIN {X 0,Y 402.932,Z 523.201,A -85,B 0,C 180,E1 -11057.623,E2 -11057.623} C_VEL
LIN {X 0,Y 402.84,Z 523.958,A -85,B 0,C 180,E1 -11058.936,E2 -11058.936} C_VEL
LIN {X 0,Y 402.772,Z 523.736,A -85,B 0,C 180,E1 -11060.964,E2 -11060.964} C_VEL
LIN {X 0,Y 402.837,Z 523.04,A -85,B 0,C 180,E1 -11061.977,E2 -11061.977} C_VEL
LIN {X 0,Y 403.027,Z 520.895,A -85,B 0,C 180,E1 -11063.703,E2 -11063.703} C_VEL
LIN {X 0,Y 403.082,Z 517.3,A -85,B 0,C 180,E1 -11065.499,E2 -11065.499} C_VEL
LIN {X 0,Y 403.354,Z 513.15,A -85,B 0,C 180,E1 -11067.003,E2 -11067.003} C_VEL
LIN {X 0,Y 403.729,Z 506.839,A -85,B 0,C 180,E1 -11068.753,E2 -11068.753} C_VEL
LIN {X 0,Y 404.272,Z 499.747,A -85,B 0,C 180,E1 -11070.29,E2 -11070.29} C_VEL
LIN {X 0,Y 403.874,Z 496.243,A -85,B 0,C 180,E1 -11070.956,E2 -11070.956} C_VEL
LIN {X 0,Y 401.425,Z 490.177,A -85,B 0,C 180,E1 -11072.028,E2 -11072.028} C_VEL
LIN {X 0,Y 399.019,Z 483.664,A -85,B 0,C 180,E1 -11073.043,E2 -11073.043} C_VEL
LIN {X 0,Y 398.685,Z 479.284,A -85,B 0,C 180,E1 -11073.61,E2 -11073.61} C_VEL
LIN {X 0,Y 399.517,Z 468.24,A -85,B 0,C 180,E1 -11074.793,E2 -11074.793} C_VEL
LIN {X 0,Y 400.345,Z 457.955,A -85,B 0,C 180,E1 -11075.666,E2 -11075.666} C_VEL
LIN {X 0,Y 400.987,Z 445.727,A -85,B 0,C 180,E1 -11076.478,E2 -11076.478} C_VEL
LIN {X 0,Y 401.363,Z 432.203,A -85,B 0,C 180,E1 -11077.135,E2 -11077.135} C_VEL
LIN {X 0,Y 401.852,Z 419.076,A -85,B 0,C 180,E1 -11077.536,E2 -11077.536} C_VEL
LIN {X 0,Y 402.946,Z 334.691,A -85,B 0,C 180,E1 -11079.048,E2 -11079.048} C_VEL
LIN {X 0,Y 398.98,Z 313.15,A -85,B 0,C 180,E1 -11079.638,E2 -11079.638} C_VEL
LIN {X 0,Y 398.431,Z 307.579,A -85,B 0,C 180,E1 -11080.93,E2 -11080.93} C_VEL
LIN {X 0,Y 397.25,Z 301.005,A -85,B 0,C 180,E1 -11082.507,E2 -11082.507} C_VEL
LIN {X 0,Y 397.162,Z 301.015,A -85,B 0,C 180,E1 -11086.446,E2 -11086.446} C_VEL
LIN {X 0,Y 397.144,Z 301.011,A -85,B 0,C 180,E1 -11089.647,E2 -11089.647} C_VEL
LIN {X 0,Y 397.108,Z 301.017,A -85,B 0,C 180,E1 -11093.031,E2 -11093.031} C_VEL
LIN {X 0,Y 397.072,Z 301.023,A -85,B 0,C 180,E1 -11096.262,E2 -11096.262} C_VEL
LIN {X 0,Y 397.095,Z 301.017,A -85,B 0,C 180,E1 -11099.862,E2 -11099.862} C_VEL
LIN {X 0,Y 397.114,Z 301.014,A -85,B 0,C 180,E1 -11103.717,E2 -11103.717} C_VEL
LIN {X 0,Y 397.087,Z 301.021,A -85,B 0,C 180,E1 -11107.208,E2 -11107.208} C_VEL
LIN {X 0,Y 397.05,Z 301.024,A -85,B 0,C 180,E1 -11110.437,E2 -11110.437} C_VEL
LIN {X 0,Y 397.092,Z 301.018,A -85,B 0,C 180,E1 -11113.648,E2 -11113.648} C_VEL
LIN {X 0,Y 397.095,Z 301.018,A -85,B 0,C 180,E1 -11116.521,E2 -11116.521} C_VEL
LIN {X 0,Y 397.084,Z 301.018,A -85,B 0,C 180,E1 -11120.419,E2 -11120.419} C_VEL
LIN {X 0,Y 397.091,Z 301.021,A -85,B 0,C 180,E1 -11123.004,E2 -11123.004} C_VEL
LIN {X 0,Y 397.111,Z 301.015,A -85,B 0,C 180,E1 -11126.282,E2 -11126.282} C_VEL
LIN {X 0,Y 397.097,Z 301.017,A -85,B 0,C 180,E1 -11130.135,E2 -11130.135} C_VEL
LIN {X 0,Y 397.186,Z 301.005,A -85,B 0,C 180,E1 -11132.609,E2 -11132.609} C_VEL
LIN {X 0,Y 397.118,Z 301.018,A -85,B 0,C 180,E1 -11135.981,E2 -11135.981} C_VEL
LIN {X 0,Y 397.131,Z 301.019,A -85,B 0,C 180,E1 -11139.704,E2 -11139.704} C_VEL
LIN {X 0,Y 397.176,Z 301.006,A -85,B 0,C 180,E1 -11142.844,E2 -11142.844} C_VEL
LIN {X 0,Y 397.17,Z 301.011,A -85,B 0,C 180,E1 -11145.657,E2 -11145.657} C_VEL
LIN {X 0,Y 397.19,Z 301.005,A -85,B 0,C 180,E1 -11148.777,E2 -11148.777} C_VEL
LIN {X 0,Y 397.301,Z 300.998,A -85,B 0,C 180,E1 -11152.129,E2 -11152.129} C_VEL
LIN {X 0,Y 397.241,Z 300.999,A -85,B 0,C 180,E1 -11154.925,E2 -11154.925} C_VEL
LIN {X 0,Y 397.441,Z 300.977,A -85,B 0,C 180,E1 -11157.973,E2 -11157.973} C_VEL
LIN {X 0,Y 397.57,Z 300.961,A -85,B 0,C 180,E1 -11160,E2 -11160} C_VEL
LIN {X 0,Y 397.367,Z 300.984,A -85,B 0,C 180,E1 -11163.042,E2 -11163.042} C_VEL
LIN {X 0,Y 397.365,Z 300.986,A -85,B 0,C 180,E1 -11166.092,E2 -11166.092} C_VEL
LIN {X 0,Y 397.245,Z 300.999,A -85,B 0,C 180,E1 -11169.162,E2 -11169.162} C_VEL
LIN {X 0,Y 397.212,Z 301.005,A -85,B 0,C 180,E1 -11172.258,E2 -11172.258} C_VEL
LIN {X 0,Y 397.171,Z 301.008,A -85,B 0,C 180,E1 -11175.392,E2 -11175.392} C_VEL
LIN {X 0,Y 397.155,Z 301.014,A -85,B 0,C 180,E1 -11178.574,E2 -11178.574} C_VEL
LIN {X 0,Y 397.089,Z 301.017,A -85,B 0,C 180,E1 -11181.819,E2 -11181.819} C_VEL
LIN {X 0,Y 397.15,Z 301.015,A -85,B 0,C 180,E1 -11185.132,E2 -11185.132} C_VEL
LIN {X 0,Y 397.157,Z 301.009,A -85,B 0,C 180,E1 -11187.777,E2 -11187.777} C_VEL
LIN {X 0,Y 397.083,Z 301.022,A -85,B 0,C 180,E1 -11190.882,E2 -11190.882} C_VEL
LIN {X 0,Y 397.12,Z 301.014,A -85,B 0,C 180,E1 -11194.494,E2 -11194.494} C_VEL
LIN {X 0,Y 397.102,Z 301.016,A -85,B 0,C 180,E1 -11198.275,E2 -11198.275} C_VEL
LIN {X 0,Y 397.086,Z 301.02,A -85,B 0,C 180,E1 -11200.909,E2 -11200.909} C_VEL
LIN {X 0,Y 397.099,Z 301.021,A -85,B 0,C 180,E1 -11203.649,E2 -11203.649} C_VEL
LIN {X 0,Y 397.098,Z 301.016,A -85,B 0,C 180,E1 -11206.522,E2 -11206.522} C_VEL
LIN {X 0,Y 397.109,Z 301.015,A -85,B 0,C 180,E1 -11210.424,E2 -11210.424} C_VEL
LIN {X 0,Y 397.105,Z 301.017,A -85,B 0,C 180,E1 -11214.266,E2 -11214.266} C_VEL
LIN {X 0,Y 397.112,Z 301.014,A -85,B 0,C 180,E1 -11216.728,E2 -11216.728} C_VEL
LIN {X 0,Y 397.123,Z 301.018,A -85,B 0,C 180,E1 -11220.297,E2 -11220.297} C_VEL
LIN {X 0,Y 397.228,Z 301.152,A -85,B 0,C 180,E1 -11222.098,E2 -11222.098} C_VEL
LIN {X 0,Y 399.808,Z 314.566,A -85,B 0,C 180,E1 -11225.047,E2 -11225.047} C_VEL
LIN {X 0,Y 399.965,Z 319.268,A -85,B 0,C 180,E1 -11226.025,E2 -11226.025} C_VEL
LIN {X 0,Y 398.741,Z 337.192,A -85,B 0,C 180,E1 -11229.63,E2 -11229.63} C_VEL
LIN {X 0,Y 398.52,Z 340.954,A -85,B 0,C 180,E1 -11230.382,E2 -11230.382} C_VEL
LIN {X 0,Y 402.592,Z 369.998,A -85,B 0,C 180,E1 -11231.089,E2 -11231.089} C_VEL
LIN {X 0,Y 401.635,Z 449.749,A -85,B 0,C 180,E1 -11232.531,E2 -11232.531} C_VEL
LIN {X 0,Y 401.132,Z 462.965,A -85,B 0,C 180,E1 -11232.968,E2 -11232.968} C_VEL
LIN {X 0,Y 400.547,Z 475.129,A -85,B 0,C 180,E1 -11233.566,E2 -11233.566} C_VEL
LIN {X 0,Y 399.785,Z 486.578,A -85,B 0,C 180,E1 -11234.32,E2 -11234.32} C_VEL
LIN {X 0,Y 398.974,Z 498.358,A -85,B 0,C 180,E1 -11235.333,E2 -11235.333} C_VEL
LIN {X 0,Y 398.223,Z 509.468,A -85,B 0,C 180,E1 -11236.541,E2 -11236.541} C_VEL
LIN {X 0,Y 397.565,Z 518.458,A -85,B 0,C 180,E1 -11237.753,E2 -11237.753} C_VEL
LIN {X 0,Y 396.802,Z 527.609,A -85,B 0,C 180,E1 -11239.283,E2 -11239.283} C_VEL
LIN {X 0,Y 396.355,Z 534.986,A -85,B 0,C 180,E1 -11240.818,E2 -11240.818} C_VEL
LIN {X 0,Y 396.057,Z 540.892,A -85,B 0,C 180,E1 -11242.353,E2 -11242.353} C_VEL
LIN {X 0,Y 395.825,Z 546.317,A -85,B 0,C 180,E1 -11244.199,E2 -11244.199} C_VEL
LIN {X 0,Y 395.78,Z 549.981,A -85,B 0,C 180,E1 -11245.927,E2 -11245.927} C_VEL
LIN {X 0,Y 395.76,Z 551.561,A -85,B 0,C 180,E1 -11246.947,E2 -11246.947} C_VEL
LIN {X 0,Y 395.825,Z 552.717,A -85,B 0,C 180,E1 -11247.966,E2 -11247.966} C_VEL
LIN {X 0,Y 395.81,Z 553.432,A -85,B 0,C 180,E1 -11248.983,E2 -11248.983} C_VEL
LIN {X 0,Y 395.797,Z 553.76,A -85,B 0,C 180,E1 -11250.001,E2 -11250.001} C_VEL
LIN {X 0,Y 395.795,Z 553.701,A -85,B 0,C 180,E1 -11251.018,E2 -11251.018} C_VEL
LIN {X 0,Y 395.804,Z 553.244,A -85,B 0,C 180,E1 -11252.036,E2 -11252.036} C_VEL
LIN {X 0,Y 395.776,Z 551.067,A -85,B 0,C 180,E1 -11254.074,E2 -11254.074} C_VEL
LIN {X 0,Y 395.827,Z 547.932,A -85,B 0,C 180,E1 -11255.805,E2 -11255.805} C_VEL
LIN {X 0,Y 396.069,Z 543.176,A -85,B 0,C 180,E1 -11257.648,E2 -11257.648} C_VEL
LIN {X 0,Y 396.505,Z 536.938,A -85,B 0,C 180,E1 -11259.437,E2 -11259.437} C_VEL
LIN {X 0,Y 397.057,Z 530.169,A -85,B 0,C 180,E1 -11260.969,E2 -11260.969} C_VEL
LIN {X 0,Y 398.013,Z 521.786,A -85,B 0,C 180,E1 -11262.493,E2 -11262.493} C_VEL
LIN {X 0,Y 398.803,Z 513.17,A -85,B 0,C 180,E1 -11263.763,E2 -11263.763} C_VEL
LIN {X 0,Y 399.551,Z 504.108,A -85,B 0,C 180,E1 -11264.868,E2 -11264.868} C_VEL
LIN {X 0,Y 400.55,Z 493.521,A -85,B 0,C 180,E1 -11265.912,E2 -11265.912} C_VEL
LIN {X 0,Y 401.5,Z 482.343,A -85,B 0,C 180,E1 -11266.788,E2 -11266.788} C_VEL
LIN {X 0,Y 402.425,Z 469.815,A -85,B 0,C 180,E1 -11267.533,E2 -11267.533} C_VEL
LIN {X 0,Y 403.164,Z 456.441,A -85,B 0,C 180,E1 -11268.09,E2 -11268.09} C_VEL
LIN {X 0,Y 403.56,Z 444.093,A -85,B 0,C 180,E1 -11268.415,E2 -11268.415} C_VEL
LIN {X 0,Y 404.62,Z 370.41,A -85,B 0,C 180,E1 -11269.745,E2 -11269.745} C_VEL
LIN {X 0,Y 400.988,Z 348.632,A -85,B 0,C 180,E1 -11270.374,E2 -11270.374} C_VEL
LIN {X 0,Y 399.392,Z 340.4,A -85,B 0,C 180,E1 -11270.662,E2 -11270.662} C_VEL
LIN {X 0,Y 400.879,Z 322.836,A -85,B 0,C 180,E1 -11274.267,E2 -11274.267} C_VEL
LIN {X 0,Y 400.908,Z 318.657,A -85,B 0,C 180,E1 -11275.158,E2 -11275.158} C_VEL
LIN {X 0,Y 398.775,Z 307.818,A -85,B 0,C 180,E1 -11277.666,E2 -11277.666} C_VEL
LIN {X 0,Y 397.151,Z 301.021,A -85,B 0,C 180,E1 -11279.338,E2 -11279.338} C_VEL
LIN {X 0,Y 397.117,Z 301.015,A -85,B 0,C 180,E1 -11283.273,E2 -11283.273} C_VEL
LIN {X 0,Y 397.11,Z 301.02,A -85,B 0,C 180,E1 -11285.735,E2 -11285.735} C_VEL
LIN {X 0,Y 397.114,Z 301.018,A -85,B 0,C 180,E1 -11289.577,E2 -11289.577} C_VEL
LIN {X 0,Y 397.103,Z 301.018,A -85,B 0,C 180,E1 -11293.479,E2 -11293.479} C_VEL
LIN {X 0,Y 397.103,Z 301.021,A -85,B 0,C 180,E1 -11296.521,E2 -11296.521} C_VEL
LIN {X 0,Y 397.114,Z 301.015,A -85,B 0,C 180,E1 -11300.423,E2 -11300.423} C_VEL
LIN {X 0,Y 397.108,Z 301.016,A -85,B 0,C 180,E1 -11304.265,E2 -11304.265} C_VEL
LIN {X 0,Y 397.115,Z 301.015,A -85,B 0,C 180,E1 -11306.727,E2 -11306.727} C_VEL
LIN {X 0,Y 397.124,Z 301.012,A -85,B 0,C 180,E1 -11310.296,E2 -11310.296} C_VEL
LIN {X 0,Y 397.194,Z 301.006,A -85,B 0,C 180,E1 -11312.61,E2 -11312.61} C_VEL
LIN {X 0,Y 397.132,Z 301.012,A -85,B 0,C 180,E1 -11315.982,E2 -11315.982} C_VEL
LIN {X 0,Y 397.138,Z 301.014,A -85,B 0,C 180,E1 -11319.704,E2 -11319.704} C_VEL
LIN {X 0,Y 397.181,Z 301.006,A -85,B 0,C 180,E1 -11322.845,E2 -11322.845} C_VEL
LIN {X 0,Y 397.228,Z 300.997,A -85,B 0,C 180,E1 -11326.703,E2 -11326.703} C_VEL
LIN {X 0,Y 397.217,Z 300.999,A -85,B 0,C 180,E1 -11329.809,E2 -11329.809} C_VEL
LIN {X 0,Y 397.351,Z 300.982,A -85,B 0,C 180,E1 -11332.888,E2 -11332.888} C_VEL
LIN {X 0,Y 397.253,Z 300.99,A -85,B 0,C 180,E1 -11334.925,E2 -11334.925} C_VEL
LIN {X 0,Y 397.448,Z 300.971,A -85,B 0,C 180,E1 -11337.973,E2 -11337.973} C_VEL
LIN {X 0,Y 397.577,Z 300.955,A -85,B 0,C 180,E1 -11340,E2 -11340} C_VEL
LIN {X 0,Y 397.374,Z 300.975,A -85,B 0,C 180,E1 -11343.041,E2 -11343.041} C_VEL
LIN {X 0,Y 397.361,Z 300.979,A -85,B 0,C 180,E1 -11347.112,E2 -11347.112} C_VEL
LIN {X 0,Y 397.216,Z 301.006,A -85,B 0,C 180,E1 -11350.191,E2 -11350.191} C_VEL
LIN {X 0,Y 397.226,Z 300.999,A -85,B 0,C 180,E1 -11353.321,E2 -11353.321} C_VEL
LIN {X 0,Y 397.181,Z 301.007,A -85,B 0,C 180,E1 -11357.155,E2 -11357.155} C_VEL
LIN {X 0,Y 397.101,Z 301.017,A -85,B 0,C 180,E1 -11360.73,E2 -11360.73} C_VEL
LIN {X 0,Y 397.128,Z 301.012,A -85,B 0,C 180,E1 -11364.018,E2 -11364.018} C_VEL
LIN {X 0,Y 397.193,Z 301.003,A -85,B 0,C 180,E1 -11367.39,E2 -11367.39} C_VEL
LIN {X 0,Y 397.078,Z 301.021,A -85,B 0,C 180,E1 -11370.882,E2 -11370.882} C_VEL
LIN {X 0,Y 397.124,Z 301.013,A -85,B 0,C 180,E1 -11374.493,E2 -11374.493} C_VEL
LIN {X 0,Y 397.1,Z 301.016,A -85,B 0,C 180,E1 -11378.275,E2 -11378.275} C_VEL
LIN {X 0,Y 397.088,Z 301.019,A -85,B 0,C 180,E1 -11380.909,E2 -11380.909} C_VEL
LIN {X 0,Y 397.101,Z 301.022,A -85,B 0,C 180,E1 -11383.648,E2 -11383.648} C_VEL
LIN {X 0,Y 397.102,Z 301.018,A -85,B 0,C 180,E1 -11386.521,E2 -11386.521} C_VEL
LIN {X 0,Y 397.113,Z 301.019,A -85,B 0,C 180,E1 -11390.423,E2 -11390.423} C_VEL
LIN {X 0,Y 397.108,Z 301.017,A -85,B 0,C 180,E1 -11394.265,E2 -11394.265} C_VEL
LIN {X 0,Y 397.152,Z 301.186,A -85,B 0,C 180,E1 -11396.375,E2 -11396.375} C_VEL
LIN {X 0,Y 399.428,Z 311.776,A -85,B 0,C 180,E1 -11399.025,E2 -11399.025} C_VEL
LIN {X 0,Y 399.755,Z 313.697,A -85,B 0,C 180,E1 -11399.437,E2 -11399.437} C_VEL
LIN {X 0,Y 402.996,Z 325.761,A -85,B 0,C 180,E1 -11399.869,E2 -11399.869} C_VEL
LIN {X 0,Y 405.051,Z 335.285,A -85,B 0,C 180,E1 -11400.175,E2 -11400.175} C_VEL
LIN {X 0,Y 403.652,Z 421.352,A -85,B 0,C 180,E1 -11401.747,E2 -11401.747} C_VEL
LIN {X 0,Y 403.11,Z 435.192,A -85,B 0,C 180,E1 -11402.219,E2 -11402.219} C_VEL
LIN {X 0,Y 402.581,Z 447.93,A -85,B 0,C 180,E1 -11402.88,E2 -11402.88} C_VEL
LIN {X 0,Y 401.82,Z 459.061,A -85,B 0,C 180,E1 -11403.652,E2 -11403.652} C_VEL
LIN {X 0,Y 400.859,Z 470.825,A -85,B 0,C 180,E1 -11404.7,E2 -11404.7} C_VEL
LIN {X 0,Y 399.912,Z 481.547,A -85,B 0,C 180,E1 -11405.911,E2 -11405.911} C_VEL
LIN {X 0,Y 398.964,Z 490.703,A -85,B 0,C 180,E1 -11407.198,E2 -11407.198} C_VEL
LIN {X 0,Y 398.204,Z 498.379,A -85,B 0,C 180,E1 -11408.517,E2 -11408.517} C_VEL
LIN {X 0,Y 397.518,Z 505.05,A -85,B 0,C 180,E1 -11409.911,E2 -11409.911} C_VEL
LIN {X 0,Y 396.918,Z 510.878,A -85,B 0,C 180,E1 -11411.414,E2 -11411.414} C_VEL
LIN {X 0,Y 396.451,Z 516.251,A -85,B 0,C 180,E1 -11413.191,E2 -11413.191} C_VEL
LIN {X 0,Y 396.165,Z 519.372,A -85,B 0,C 180,E1 -11414.567,E2 -11414.567} C_VEL
LIN {X 0,Y 395.961,Z 521.239,A -85,B 0,C 180,E1 -11415.612,E2 -11415.612} C_VEL
LIN {X 0,Y 395.841,Z 523.483,A -85,B 0,C 180,E1 -11417.555,E2 -11417.555} C_VEL
LIN {X 0,Y 395.753,Z 524.172,A -85,B 0,C 180,E1 -11418.735,E2 -11418.735} C_VEL
LIN {X 0,Y 395.68,Z 524.331,A -85,B 0,C 180,E1 -11419.769,E2 -11419.769} C_VEL
LIN {X 0,Y 395.751,Z 523.41,A -85,B 0,C 180,E1 -11421.832,E2 -11421.832} C_VEL
LIN {X 0,Y 395.944,Z 521.165,A -85,B 0,C 180,E1 -11423.719,E2 -11423.719} C_VEL
LIN {X 0,Y 396.003,Z 517.884,A -85,B 0,C 180,E1 -11425.419,E2 -11425.419} C_VEL
LIN {X 0,Y 396.271,Z 513.83,A -85,B 0,C 180,E1 -11426.95,E2 -11426.95} C_VEL
LIN {X 0,Y 396.618,Z 507.625,A -85,B 0,C 180,E1 -11428.73,E2 -11428.73} C_VEL
LIN {X 0,Y 397.168,Z 500.868,A -85,B 0,C 180,E1 -11430.253,E2 -11430.253} C_VEL
LIN {X 0,Y 397.818,Z 492.469,A -85,B 0,C 180,E1 -11431.771,E2 -11431.771} C_VEL
LIN {X 0,Y 398.37,Z 483.855,A -85,B 0,C 180,E1 -11433.033,E2 -11433.033} C_VEL
LIN {X 0,Y 398.685,Z 479.284,A -85,B 0,C 180,E1 -11433.61,E2 -11433.61} C_VEL
LIN {X 0,Y 398.403,Z 474.779,A -85,B 0,C 180,E1 -11434.148,E2 -11434.148} C_VEL
LIN {X 0,Y 396.237,Z 467.198,A -85,B 0,C 180,E1 -11435.009,E2 -11435.009} C_VEL
LIN {X 0,Y 394.035,Z 459.169,A -85,B 0,C 180,E1 -11435.796,E2 -11435.796} C_VEL
LIN {X 0,Y 393.705,Z 453.903,A -85,B 0,C 180,E1 -11436.213,E2 -11436.213} C_VEL
LIN {X 0,Y 394.314,Z 441.435,A -85,B 0,C 180,E1 -11436.974,E2 -11436.974} C_VEL
LIN {X 0,Y 394.583,Z 429.097,A -85,B 0,C 180,E1 -11437.515,E2 -11437.515} C_VEL
LIN {X 0,Y 395.039,Z 417.893,A -85,B 0,C 180,E1 -11437.828,E2 -11437.828} C_VEL
LIN {X 0,Y 396.102,Z 335.419,A -85,B 0,C 180,E1 -11439.327,E2 -11439.327} C_VEL
LIN {X 0,Y 392.025,Z 313.463,A -85,B 0,C 180,E1 -11439.93,E2 -11439.93} C_VEL
LIN {X 0,Y 390.84,Z 305.081,A -85,B 0,C 180,E1 -11441.934,E2 -11441.934} C_VEL
LIN {X 0,Y 390.222,Z 301.88,A -85,B 0,C 180,E1 -11442.761,E2 -11442.761} C_VEL
LIN {X 0,Y 390.135,Z 301.886,A -85,B 0,C 180,E1 -11446.751,E2 -11446.751} C_VEL
LIN {X 0,Y 390.086,Z 301.897,A -85,B 0,C 180,E1 -11450.469,E2 -11450.469} C_VEL
LIN {X 0,Y 390.06,Z 301.893,A -85,B 0,C 180,E1 -11453.352,E2 -11453.352} C_VEL
LIN {X 0,Y 390.027,Z 301.903,A -85,B 0,C 180,E1 -11456.774,E2 -11456.774} C_VEL
LIN {X 0,Y 390.033,Z 301.899,A -85,B 0,C 180,E1 -11460.299,E2 -11460.299} C_VEL
LIN {X 0,Y 390.064,Z 301.893,A -85,B 0,C 180,E1 -11464.024,E2 -11464.024} C_VEL
LIN {X 0,Y 390.036,Z 301.897,A -85,B 0,C 180,E1 -11467.549,E2 -11467.549} C_VEL
LIN {X 0,Y 390.013,Z 301.904,A -85,B 0,C 180,E1 -11470.814,E2 -11470.814} C_VEL
LIN {X 0,Y 390.046,Z 301.895,A -85,B 0,C 180,E1 -11473.885,E2 -11473.885} C_VEL
LIN {X 0,Y 390.049,Z 301.897,A -85,B 0,C 180,E1 -11476.789,E2 -11476.789} C_VEL
LIN {X 0,Y 390.049,Z 301.898,A -85,B 0,C 180,E1 -11479.56,E2 -11479.56} C_VEL
LIN {X 0,Y 390.034,Z 301.896,A -85,B 0,C 180,E1 -11482.449,E2 -11482.449} C_VEL
LIN {X 0,Y 390.061,Z 301.894,A -85,B 0,C 180,E1 -11485.975,E2 -11485.975} C_VEL
LIN {X 0,Y 390.039,Z 301.899,A -85,B 0,C 180,E1 -11489.869,E2 -11489.869} C_VEL
LIN {X 0,Y 390.104,Z 301.891,A -85,B 0,C 180,E1 -11493.231,E2 -11493.231} C_VEL
LIN {X 0,Y 390.059,Z 301.893,A -85,B 0,C 180,E1 -11496.763,E2 -11496.763} C_VEL
LIN {X 0,Y 390.096,Z 301.893,A -85,B 0,C 180,E1 -11499.983,E2 -11499.983} C_VEL
LIN {X 0,Y 390.133,Z 301.885,A -85,B 0,C 180,E1 -11503.248,E2 -11503.248} C_VEL
LIN {X 0,Y 390.186,Z 301.878,A -85,B 0,C 180,E1 -11506.561,E2 -11506.561} C_VEL
LIN {X 0,Y 390.195,Z 301.877,A -85,B 0,C 180,E1 -11510.671,E2 -11510.671} C_VEL
LIN {X 0,Y 390.299,Z 301.866,A -85,B 0,C 180,E1 -11513.798,E2 -11513.798} C_VEL
LIN {X 0,Y 390.41,Z 301.853,A -85,B 0,C 180,E1 -11517.937,E2 -11517.937} C_VEL
LIN {X 0,Y 390.539,Z 301.837,A -85,B 0,C 180,E1 -11520,E2 -11520} C_VEL
LIN {X 0,Y 390.302,Z 301.863,A -85,B 0,C 180,E1 -11523.097,E2 -11523.097} C_VEL
LIN {X 0,Y 390.319,Z 301.865,A -85,B 0,C 180,E1 -11526.202,E2 -11526.202} C_VEL
LIN {X 0,Y 390.197,Z 301.876,A -85,B 0,C 180,E1 -11529.329,E2 -11529.329} C_VEL
LIN {X 0,Y 390.187,Z 301.878,A -85,B 0,C 180,E1 -11533.439,E2 -11533.439} C_VEL
LIN {X 0,Y 390.141,Z 301.885,A -85,B 0,C 180,E1 -11537.308,E2 -11537.308} C_VEL
LIN {X 0,Y 390.08,Z 301.893,A -85,B 0,C 180,E1 -11540.471,E2 -11540.471} C_VEL
LIN {X 0,Y 390.082,Z 301.893,A -85,B 0,C 180,E1 -11543.351,E2 -11543.351} C_VEL
LIN {X 0,Y 390.107,Z 301.891,A -85,B 0,C 180,E1 -11546.769,E2 -11546.769} C_VEL
LIN {X 0,Y 390.04,Z 301.896,A -85,B 0,C 180,E1 -11550.3,E2 -11550.3} C_VEL
LIN {X 0,Y 390.05,Z 301.896,A -85,B 0,C 180,E1 -11552.721,E2 -11552.721} C_VEL
LIN {X 0,Y 390.052,Z 301.896,A -85,B 0,C 180,E1 -11555.826,E2 -11555.826} C_VEL
LIN {X 0,Y 390.067,Z 301.898,A -85,B 0,C 180,E1 -11559.22,E2 -11559.22} C_VEL
LIN {X 0,Y 390.04,Z 301.895,A -85,B 0,C 180,E1 -11562.375,E2 -11562.375} C_VEL
LIN {X 0,Y 390.042,Z 301.901,A -85,B 0,C 180,E1 -11565.356,E2 -11565.356} C_VEL
LIN {X 0,Y 390.027,Z 301.898,A -85,B 0,C 180,E1 -11568.188,E2 -11568.188} C_VEL
LIN {X 0,Y 390.084,Z 301.89,A -85,B 0,C 180,E1 -11570.908,E2 -11570.908} C_VEL
LIN {X 0,Y 390.083,Z 301.89,A -85,B 0,C 180,E1 -11574.794,E2 -11574.794} C_VEL
LIN {X 0,Y 390.022,Z 301.899,A -85,B 0,C 180,E1 -11578.497,E2 -11578.497} C_VEL
LIN {X 0,Y 390.175,Z 301.97,A -85,B 0,C 180,E1 -11581.853,E2 -11581.853} C_VEL
LIN {X 0,Y 392.994,Z 316.705,A -85,B 0,C 180,E1 -11585.15,E2 -11585.15} C_VEL
LIN {X 0,Y 392.861,Z 322.058,A -85,B 0,C 180,E1 -11586.266,E2 -11586.266} C_VEL
LIN {X 0,Y 391.742,Z 337.982,A -85,B 0,C 180,E1 -11589.524,E2 -11589.524} C_VEL
LIN {X 0,Y 391.546,Z 340.626,A -85,B 0,C 180,E1 -11590.061,E2 -11590.061} C_VEL
LIN {X 0,Y 395.79,Z 371.41,A -85,B 0,C 180,E1 -11590.834,E2 -11590.834} C_VEL
LIN {X 0,Y 394.812,Z 448.867,A -85,B 0,C 180,E1 -11592.252,E2 -11592.252} C_VEL
LIN {X 0,Y 394.248,Z 462.289,A -85,B 0,C 180,E1 -11592.695,E2 -11592.695} C_VEL
LIN {X 0,Y 393.639,Z 475.138,A -85,B 0,C 180,E1 -11593.336,E2 -11593.336} C_VEL
LIN {X 0,Y 392.791,Z 487.311,A -85,B 0,C 180,E1 -11594.166,E2 -11594.166} C_VEL
LIN {X 0,Y 391.959,Z 498.902,A -85,B 0,C 180,E1 -11595.197,E2 -11595.197} C_VEL
LIN {X 0,Y 391.257,Z 509.048,A -85,B 0,C 180,E1 -11596.327,E2 -11596.327} C_VEL
LIN {X 0,Y 390.568,Z 517.872,A -85,B 0,C 180,E1 -11597.531,E2 -11597.531} C_VEL
LIN {X 0,Y 389.797,Z 527.091,A -85,B 0,C 180,E1 -11599.088,E2 -11599.088} C_VEL
LIN {X 0,Y 389.326,Z 534.515,A -85,B 0,C 180,E1 -11600.651,E2 -11600.651} C_VEL
LIN {X 0,Y 388.986,Z 540.46,A -85,B 0,C 180,E1 -11602.213,E2 -11602.213} C_VEL
LIN {X 0,Y 388.774,Z 545.362,A -85,B 0,C 180,E1 -11603.857,E2 -11603.857} C_VEL
LIN {X 0,Y 388.719,Z 548.697,A -85,B 0,C 180,E1 -11605.334,E2 -11605.334} C_VEL
LIN {X 0,Y 388.664,Z 551.231,A -85,B 0,C 180,E1 -11606.891,E2 -11606.891} C_VEL
LIN {X 0,Y 388.724,Z 552.412,A -85,B 0,C 180,E1 -11607.928,E2 -11607.928} C_VEL
LIN {X 0,Y 388.74,Z 553.147,A -85,B 0,C 180,E1 -11608.965,E2 -11608.965} C_VEL
LIN {X 0,Y 388.726,Z 553.488,A -85,B 0,C 180,E1 -11610.001,E2 -11610.001} C_VEL
LIN {X 0,Y 388.726,Z 553.444,A -85,B 0,C 180,E1 -11611.036,E2 -11611.036} C_VEL
LIN {X 0,Y 388.701,Z 553.008,A -85,B 0,C 180,E1 -11612.073,E2 -11612.073} C_VEL
LIN {X 0,Y 388.701,Z 550.868,A -85,B 0,C 180,E1 -11614.148,E2 -11614.148} C_VEL
LIN {X 0,Y 388.775,Z 547.28,A -85,B 0,C 180,E1 -11616.144,E2 -11616.144} C_VEL
LIN {X 0,Y 389.022,Z 543.055,A -85,B 0,C 180,E1 -11617.788,E2 -11617.788} C_VEL
LIN {X 0,Y 389.485,Z 536.86,A -85,B 0,C 180,E1 -11619.609,E2 -11619.609} C_VEL
LIN {X 0,Y 390.062,Z 530.133,A -85,B 0,C 180,E1 -11621.169,E2 -11621.169} C_VEL
LIN {X 0,Y 391.069,Z 521.815,A -85,B 0,C 180,E1 -11622.718,E2 -11622.718} C_VEL
LIN {X 0,Y 391.967,Z 512.088,A -85,B 0,C 180,E1 -11624.17,E2 -11624.17} C_VEL
LIN {X 0,Y 392.937,Z 501.726,A -85,B 0,C 180,E1 -11625.417,E2 -11625.417} C_VEL
LIN {X 0,Y 394.011,Z 490.967,A -85,B 0,C 180,E1 -11626.449,E2 -11626.449} C_VEL
LIN {X 0,Y 395.071,Z 479.064,A -85,B 0,C 180,E1 -11627.336,E2 -11627.336} C_VEL
LIN {X 0,Y 395.966,Z 466.703,A -85,B 0,C 180,E1 -11628.029,E2 -11628.029} C_VEL
LIN {X 0,Y 396.716,Z 453.959,A -85,B 0,C 180,E1 -11628.528,E2 -11628.528} C_VEL
LIN {X 0,Y 397.054,Z 440.112,A -85,B 0,C 180,E1 -11628.855,E2 -11628.855} C_VEL
LIN {X 0,Y 397.994,Z 370.779,A -85,B 0,C 180,E1 -11630.131,E2 -11630.131} C_VEL
LIN {X 0,Y 393.936,Z 347.003,A -85,B 0,C 180,E1 -11630.842,E2 -11630.842} C_VEL
LIN {X 0,Y 392.537,Z 340.2,A -85,B 0,C 180,E1 -11631.082,E2 -11631.082} C_VEL
LIN {X 0,Y 393.878,Z 325.133,A -85,B 0,C 180,E1 -11634.23,E2 -11634.23} C_VEL
LIN {X 0,Y 394.137,Z 321.08,A -85,B 0,C 180,E1 -11635.093,E2 -11635.093} C_VEL
LIN {X 0,Y 392.209,Z 310.918,A -85,B 0,C 180,E1 -11637.478,E2 -11637.478} C_VEL
LIN {X 0,Y 390.081,Z 301.902,A -85,B 0,C 180,E1 -11639.7,E2 -11639.7} C_VEL
LIN {X 0,Y 390.045,Z 301.896,A -85,B 0,C 180,E1 -11642.721,E2 -11642.721} C_VEL
LIN {X 0,Y 390.058,Z 301.899,A -85,B 0,C 180,E1 -11645.825,E2 -11645.825} C_VEL
LIN {X 0,Y 390.068,Z 301.895,A -85,B 0,C 180,E1 -11649.218,E2 -11649.218} C_VEL
LIN {X 0,Y 390.043,Z 301.9,A -85,B 0,C 180,E1 -11652.374,E2 -11652.374} C_VEL
LIN {X 0,Y 390.045,Z 301.898,A -85,B 0,C 180,E1 -11655.354,E2 -11655.354} C_VEL
LIN {X 0,Y 390.032,Z 301.899,A -85,B 0,C 180,E1 -11658.186,E2 -11658.186} C_VEL
LIN {X 0,Y 390.089,Z 301.895,A -85,B 0,C 180,E1 -11660.907,E2 -11660.907} C_VEL
LIN {X 0,Y 390.085,Z 301.896,A -85,B 0,C 180,E1 -11664.793,E2 -11664.793} C_VEL
LIN {X 0,Y 390.024,Z 301.9,A -85,B 0,C 180,E1 -11668.495,E2 -11668.495} C_VEL
LIN {X 0,Y 390.117,Z 301.886,A -85,B 0,C 180,E1 -11672.07,E2 -11672.07} C_VEL
LIN {X 0,Y 390.08,Z 301.895,A -85,B 0,C 180,E1 -11675.519,E2 -11675.519} C_VEL
LIN {X 0,Y 390.055,Z 301.896,A -85,B 0,C 180,E1 -11678.878,E2 -11678.878} C_VEL
LIN {X 0,Y 390.128,Z 301.884,A -85,B 0,C 180,E1 -11682.167,E2 -11682.167} C_VEL
LIN {X 0,Y 390.144,Z 301.882,A -85,B 0,C 180,E1 -11685.392,E2 -11685.392} C_VEL
LIN {X 0,Y 390.146,Z 301.88,A -85,B 0,C 180,E1 -11688.571,E2 -11688.571} C_VEL
LIN {X 0,Y 390.307,Z 301.864,A -85,B 0,C 180,E1 -11692.032,E2 -11692.032} C_VEL
LIN {X 0,Y 390.225,Z 301.865,A -85,B 0,C 180,E1 -11694.833,E2 -11694.833} C_VEL
LIN {X 0,Y 390.417,Z 301.847,A -85,B 0,C 180,E1 -11697.937,E2 -11697.937} C_VEL
LIN {X 0,Y 390.547,Z 301.83,A -85,B 0,C 180,E1 -11700,E2 -11700} C_VEL
LIN {X 0,Y 390.309,Z 301.855,A -85,B 0,C 180,E1 -11703.096,E2 -11703.096} C_VEL
LIN {X 0,Y 390.306,Z 301.86,A -85,B 0,C 180,E1 -11706.639,E2 -11706.639} C_VEL
LIN {X 0,Y 390.204,Z 301.873,A -85,B 0,C 180,E1 -11709.329,E2 -11709.329} C_VEL
LIN {X 0,Y 390.193,Z 301.875,A -85,B 0,C 180,E1 -11713.438,E2 -11713.438} C_VEL
LIN {X 0,Y 390.148,Z 301.882,A -85,B 0,C 180,E1 -11717.308,E2 -11717.308} C_VEL
LIN {X 0,Y 390.086,Z 301.891,A -85,B 0,C 180,E1 -11720.47,E2 -11720.47} C_VEL
LIN {X 0,Y 390.072,Z 301.892,A -85,B 0,C 180,E1 -11723.352,E2 -11723.352} C_VEL
LIN {X 0,Y 390.113,Z 301.892,A -85,B 0,C 180,E1 -11726.768,E2 -11726.768} C_VEL
LIN {X 0,Y 390.038,Z 301.896,A -85,B 0,C 180,E1 -11730.3,E2 -11730.3} C_VEL
LIN {X 0,Y 390.067,Z 301.891,A -85,B 0,C 180,E1 -11734.025,E2 -11734.025} C_VEL
LIN {X 0,Y 390.042,Z 301.897,A -85,B 0,C 180,E1 -11737.551,E2 -11737.551} C_VEL
LIN {X 0,Y 390.056,Z 301.894,A -85,B 0,C 180,E1 -11740.821,E2 -11740.821} C_VEL
LIN {X 0,Y 390.054,Z 301.898,A -85,B 0,C 180,E1 -11743.886,E2 -11743.886} C_VEL
LIN {X 0,Y 390.057,Z 301.896,A -85,B 0,C 180,E1 -11746.79,E2 -11746.79} C_VEL
LIN {X 0,Y 390.056,Z 301.9,A -85,B 0,C 180,E1 -11749.56,E2 -11749.56} C_VEL
LIN {X 0,Y 390.042,Z 301.895,A -85,B 0,C 180,E1 -11752.449,E2 -11752.449} C_VEL
LIN {X 0,Y 390.091,Z 301.945,A -85,B 0,C 180,E1 -11755.97,E2 -11755.97} C_VEL
LIN {X 0,Y 392.613,Z 313.703,A -85,B 0,C 180,E1 -11758.971,E2 -11758.971} C_VEL
LIN {X 0,Y 395.127,Z 321.496,A -85,B 0,C 180,E1 -11759.293,E2 -11759.293} C_VEL
LIN {X 0,Y 398.566,Z 336.512,A -85,B 0,C 180,E1 -11759.803,E2 -11759.803} C_VEL
LIN {X 0,Y 397.05,Z 421.621,A -85,B 0,C 180,E1 -11761.379,E2 -11761.379} C_VEL
LIN {X 0,Y 396.46,Z 435.435,A -85,B 0,C 180,E1 -11761.855,E2 -11761.855} C_VEL
LIN {X 0,Y 395.915,Z 447.971,A -85,B 0,C 180,E1 -11762.514,E2 -11762.514} C_VEL
LIN {X 0,Y 395.094,Z 459.668,A -85,B 0,C 180,E1 -11763.341,E2 -11763.341} C_VEL
LIN {X 0,Y 394.113,Z 471.088,A -85,B 0,C 180,E1 -11764.377,E2 -11764.377} C_VEL
LIN {X 0,Y 393.119,Z 481.603,A -85,B 0,C 180,E1 -11765.58,E2 -11765.58} C_VEL
LIN {X 0,Y 392.216,Z 490.129,A -85,B 0,C 180,E1 -11766.783,E2 -11766.783} C_VEL
LIN {X 0,Y 391.352,Z 497.941,A -85,B 0,C 180,E1 -11768.122,E2 -11768.122} C_VEL
LIN {X 0,Y 390.612,Z 505.08,A -85,B 0,C 180,E1 -11769.623,E2 -11769.623} C_VEL
LIN {X 0,Y 389.985,Z 510.674,A -85,B 0,C 180,E1 -11771.072,E2 -11771.072} C_VEL
LIN {X 0,Y 389.494,Z 515.582,A -85,B 0,C 180,E1 -11772.67,E2 -11772.67} C_VEL
LIN {X 0,Y 389.137,Z 519.362,A -85,B 0,C 180,E1 -11774.281,E2 -11774.281} C_VEL
LIN {X 0,Y 388.928,Z 521.285,A -85,B 0,C 180,E1 -11775.346,E2 -11775.346} C_VEL
LIN {X 0,Y 388.787,Z 522.742,A -85,B 0,C 180,E1 -11776.408,E2 -11776.408} C_VEL
LIN {X 0,Y 388.77,Z 523.756,A -85,B 0,C 180,E1 -11777.471,E2 -11777.471} C_VEL
LIN {X 0,Y 388.668,Z 524.376,A -85,B 0,C 180,E1 -11778.527,E2 -11778.527} C_VEL
LIN {X 0,Y 388.612,Z 524.604,A -85,B 0,C 180,E1 -11779.58,E2 -11779.58} C_VEL
LIN {X 0,Y 388.605,Z 524.392,A -85,B 0,C 180,E1 -11780.632,E2 -11780.632} C_VEL
LIN {X 0,Y 388.761,Z 522.776,A -85,B 0,C 180,E1 -11782.73,E2 -11782.73} C_VEL
LIN {X 0,Y 388.873,Z 521.373,A -85,B 0,C 180,E1 -11783.774,E2 -11783.774} C_VEL
LIN {X 0,Y 388.927,Z 518.449,A -85,B 0,C 180,E1 -11785.335,E2 -11785.335} C_VEL
LIN {X 0,Y 389.19,Z 514.487,A -85,B 0,C 180,E1 -11786.894,E2 -11786.894} C_VEL
LIN {X 0,Y 389.515,Z 508.403,A -85,B 0,C 180,E1 -11788.707,E2 -11788.707} C_VEL
LIN {X 0,Y 390.086,Z 501.757,A -85,B 0,C 180,E1 -11790.258,E2 -11790.258} C_VEL
LIN {X 0,Y 390.762,Z 493.528,A -85,B 0,C 180,E1 -11791.803,E2 -11791.803} C_VEL
LIN {X 0,Y 391.331,Z 485.102,A -85,B 0,C 180,E1 -11793.088,E2 -11793.088} C_VEL
LIN {X 0,Y 392.113,Z 474.688,A -85,B 0,C 180,E1 -11794.368,E2 -11794.368} C_VEL
LIN {X 0,Y 392.958,Z 465.748,A -85,B 0,C 180,E1 -11795.258,E2 -11795.258} C_VEL
LIN {X 0,Y 393.705,Z 453.903,A -85,B 0,C 180,E1 -11796.213,E2 -11796.213} C_VEL
LIN {X 0,Y 393.26,Z 450.401,A -85,B 0,C 180,E1 -11796.481,E2 -11796.481} C_VEL
LIN {X 0,Y 390.832,Z 444.906,A -85,B 0,C 180,E1 -11796.925,E2 -11796.925} C_VEL
LIN {X 0,Y 388.259,Z 439.283,A -85,B 0,C 180,E1 -11797.328,E2 -11797.328} C_VEL
LIN {X 0,Y 387.591,Z 435.575,A -85,B 0,C 180,E1 -11797.528,E2 -11797.528} C_VEL
LIN {X 0,Y 387.89,Z 426.593,A -85,B 0,C 180,E1 -11797.875,E2 -11797.875} C_VEL
LIN {X 0,Y 388.289,Z 413.391,A -85,B 0,C 180,E1 -11798.194,E2 -11798.194} C_VEL
LIN {X 0,Y 389.286,Z 336.465,A -85,B 0,C 180,E1 -11799.609,E2 -11799.609} C_VEL
LIN {X 0,Y 385.022,Z 313.683,A -85,B 0,C 180,E1 -11800.256,E2 -11800.256} C_VEL
LIN {X 0,Y 383.195,Z 302.754,A -85,B 0,C 180,E1 -11802.97,E2 -11802.97} C_VEL
LIN {X 0,Y 383.076,Z 302.766,A -85,B 0,C 180,E1 -11805.973,E2 -11805.973} C_VEL
LIN {X 0,Y 383.056,Z 302.766,A -85,B 0,C 180,E1 -11809.283,E2 -11809.283} C_VEL
LIN {X 0,Y 382.987,Z 302.78,A -85,B 0,C 180,E1 -11812.665,E2 -11812.665} C_VEL
LIN {X 0,Y 382.979,Z 302.777,A -85,B 0,C 180,E1 -11816.13,E2 -11816.13} C_VEL
LIN {X 0,Y 382.972,Z 302.776,A -85,B 0,C 180,E1 -11819.7,E2 -11819.7} C_VEL
LIN {X 0,Y 382.999,Z 302.774,A -85,B 0,C 180,E1 -11823.4,E2 -11823.4} C_VEL
LIN {X 0,Y 383.027,Z 302.77,A -85,B 0,C 180,E1 -11826.163,E2 -11826.163} C_VEL
LIN {X 0,Y 382.97,Z 302.776,A -85,B 0,C 180,E1 -11829.962,E2 -11829.962} C_VEL
LIN {X 0,Y 383,Z 302.776,A -85,B 0,C 180,E1 -11832.778,E2 -11832.778} C_VEL
LIN {X 0,Y 382.99,Z 302.775,A -85,B 0,C 180,E1 -11835.788,E2 -11835.788} C_VEL
LIN {X 0,Y 382.978,Z 302.778,A -85,B 0,C 180,E1 -11838.796,E2 -11838.796} C_VEL
LIN {X 0,Y 382.989,Z 302.774,A -85,B 0,C 180,E1 -11842.096,E2 -11842.096} C_VEL
LIN {X 0,Y 383.011,Z 302.778,A -85,B 0,C 180,E1 -11845.331,E2 -11845.331} C_VEL
LIN {X 0,Y 382.975,Z 302.778,A -85,B 0,C 180,E1 -11849.081,E2 -11849.081} C_VEL
LIN {X 0,Y 383.048,Z 302.766,A -85,B 0,C 180,E1 -11852.698,E2 -11852.698} C_VEL
LIN {X 0,Y 383.041,Z 302.768,A -85,B 0,C 180,E1 -11855.039,E2 -11855.039} C_VEL
LIN {X 0,Y 382.984,Z 302.775,A -85,B 0,C 180,E1 -11858.469,E2 -11858.469} C_VEL
LIN {X 0,Y 383.081,Z 302.77,A -85,B 0,C 180,E1 -11861.827,E2 -11861.827} C_VEL
LIN {X 0,Y 383.104,Z 302.76,A -85,B 0,C 180,E1 -11865.118,E2 -11865.118} C_VEL
LIN {X 0,Y 383.089,Z 302.765,A -85,B 0,C 180,E1 -11868.358,E2 -11868.358} C_VEL
LIN {X 0,Y 383.212,Z 302.753,A -85,B 0,C 180,E1 -11872.022,E2 -11872.022} C_VEL
LIN {X 0,Y 383.183,Z 302.751,A -85,B 0,C 180,E1 -11874.738,E2 -11874.738} C_VEL
LIN {X 0,Y 383.377,Z 302.729,A -85,B 0,C 180,E1 -11877.899,E2 -11877.899} C_VEL
LIN {X 0,Y 383.508,Z 302.713,A -85,B 0,C 180,E1 -11880,E2 -11880} C_VEL
LIN {X 0,Y 383.239,Z 302.743,A -85,B 0,C 180,E1 -11883.154,E2 -11883.154} C_VEL
LIN {X 0,Y 383.275,Z 302.743,A -85,B 0,C 180,E1 -11886.317,E2 -11886.317} C_VEL
LIN {X 0,Y 383.144,Z 302.755,A -85,B 0,C 180,E1 -11889.502,E2 -11889.502} C_VEL
LIN {X 0,Y 383.118,Z 302.758,A -85,B 0,C 180,E1 -11893.537,E2 -11893.537} C_VEL
LIN {X 0,Y 383.087,Z 302.762,A -85,B 0,C 180,E1 -11897.455,E2 -11897.455} C_VEL
LIN {X 0,Y 383.021,Z 302.774,A -85,B 0,C 180,E1 -11900.648,E2 -11900.648} C_VEL
LIN {X 0,Y 383.026,Z 302.769,A -85,B 0,C 180,E1 -11903.808,E2 -11903.808} C_VEL
LIN {X 0,Y 383.073,Z 302.763,A -85,B 0,C 180,E1 -11906.124,E2 -11906.124} C_VEL
LIN {X 0,Y 383.044,Z 302.768,A -85,B 0,C 180,E1 -11908.493,E2 -11908.493} C_VEL
LIN {X 0,Y 383.003,Z 302.772,A -85,B 0,C 180,E1 -11912.428,E2 -11912.428} C_VEL
LIN {X 0,Y 383.028,Z 302.769,A -85,B 0,C 180,E1 -11916.166,E2 -11916.166} C_VEL
LIN {X 0,Y 383.005,Z 302.773,A -85,B 0,C 180,E1 -11919.959,E2 -11919.959} C_VEL
LIN {X 0,Y 383.001,Z 302.773,A -85,B 0,C 180,E1 -11922.78,E2 -11922.78} C_VEL
LIN {X 0,Y 382.994,Z 302.777,A -85,B 0,C 180,E1 -11925.79,E2 -11925.79} C_VEL
LIN {X 0,Y 382.984,Z 302.775,A -85,B 0,C 180,E1 -11928.797,E2 -11928.797} C_VEL
LIN {X 0,Y 382.995,Z 302.776,A -85,B 0,C 180,E1 -11932.098,E2 -11932.098} C_VEL
LIN {X 0,Y 383.016,Z 302.773,A -85,B 0,C 180,E1 -11935.333,E2 -11935.333} C_VEL
LIN {X 0,Y 382.981,Z 302.775,A -85,B 0,C 180,E1 -11939.082,E2 -11939.082} C_VEL
LIN {X 0,Y 383.123,Z 302.914,A -85,B 0,C 180,E1 -11941.627,E2 -11941.627} C_VEL
LIN {X 0,Y 385.7,Z 316.108,A -85,B 0,C 180,E1 -11944.647,E2 -11944.647} C_VEL
LIN {X 0,Y 386.132,Z 320.044,A -85,B 0,C 180,E1 -11945.513,E2 -11945.513} C_VEL
LIN {X 0,Y 384.729,Z 338.765,A -85,B 0,C 180,E1 -11949.413,E2 -11949.413} C_VEL
LIN {X 0,Y 384.601,Z 340.418,A -85,B 0,C 180,E1 -11949.755,E2 -11949.755} C_VEL
LIN {X 0,Y 388.987,Z 372.034,A -85,B 0,C 180,E1 -11950.557,E2 -11950.557} C_VEL
LIN {X 0,Y 387.94,Z 449.055,A -85,B 0,C 180,E1 -11951.995,E2 -11951.995} C_VEL
LIN {X 0,Y 387.363,Z 462.321,A -85,B 0,C 180,E1 -11952.445,E2 -11952.445} C_VEL
LIN {X 0,Y 386.734,Z 475.093,A -85,B 0,C 180,E1 -11953.097,E2 -11953.097} C_VEL
LIN {X 0,Y 385.897,Z 486.403,A -85,B 0,C 180,E1 -11953.876,E2 -11953.876} C_VEL
LIN {X 0,Y 385.049,Z 498.119,A -85,B 0,C 180,E1 -11954.925,E2 -11954.925} C_VEL
LIN {X 0,Y 384.345,Z 508.001,A -85,B 0,C 180,E1 -11956.032,E2 -11956.032} C_VEL
LIN {X 0,Y 383.573,Z 517.258,A -85,B 0,C 180,E1 -11957.299,E2 -11957.299} C_VEL
LIN {X 0,Y 382.895,Z 525.179,A -85,B 0,C 180,E1 -11958.621,E2 -11958.621} C_VEL
LIN {X 0,Y 382.328,Z 532.903,A -85,B 0,C 180,E1 -11960.211,E2 -11960.211} C_VEL
LIN {X 0,Y 381.907,Z 540.021,A -85,B 0,C 180,E1 -11962.068,E2 -11962.068} C_VEL
LIN {X 0,Y 381.67,Z 545.376,A -85,B 0,C 180,E1 -11963.907,E2 -11963.907} C_VEL
LIN {X 0,Y 381.631,Z 549.288,A -85,B 0,C 180,E1 -11965.776,E2 -11965.776} C_VEL
LIN {X 0,Y 381.624,Z 552.102,A -85,B 0,C 180,E1 -11967.89,E2 -11967.89} C_VEL
LIN {X 0,Y 381.672,Z 552.86,A -85,B 0,C 180,E1 -11968.945,E2 -11968.945} C_VEL
LIN {X 0,Y 381.656,Z 553.217,A -85,B 0,C 180,E1 -11970.001,E2 -11970.001} C_VEL
LIN {X 0,Y 381.639,Z 553.186,A -85,B 0,C 180,E1 -11971.056,E2 -11971.056} C_VEL
LIN {X 0,Y 381.598,Z 552.77,A -85,B 0,C 180,E1 -11972.111,E2 -11972.111} C_VEL
LIN {X 0,Y 381.549,Z 551.924,A -85,B 0,C 180,E1 -11973.168,E2 -11973.168} C_VEL
LIN {X 0,Y 381.626,Z 550.671,A -85,B 0,C 180,E1 -11974.225,E2 -11974.225} C_VEL
LIN {X 0,Y 381.679,Z 547.428,A -85,B 0,C 180,E1 -11976.106,E2 -11976.106} C_VEL
LIN {X 0,Y 381.95,Z 542.933,A -85,B 0,C 180,E1 -11977.933,E2 -11977.933} C_VEL
LIN {X 0,Y 382.469,Z 536.792,A -85,B 0,C 180,E1 -11979.787,E2 -11979.787} C_VEL
LIN {X 0,Y 383.082,Z 530.113,A -85,B 0,C 180,E1 -11981.375,E2 -11981.375} C_VEL
LIN {X 0,Y 384.128,Z 521.848,A -85,B 0,C 180,E1 -11982.952,E2 -11982.952} C_VEL
LIN {X 0,Y 385.025,Z 512.692,A -85,B 0,C 180,E1 -11984.365,E2 -11984.365} C_VEL
LIN {X 0,Y 386.117,Z 501.927,A -85,B 0,C 180,E1 -11985.696,E2 -11985.696} C_VEL
LIN {X 0,Y 387.227,Z 491.278,A -85,B 0,C 180,E1 -11986.746,E2 -11986.746} C_VEL
LIN {X 0,Y 388.34,Z 479.589,A -85,B 0,C 180,E1 -11987.646,E2 -11987.646} C_VEL
LIN {X 0,Y 389.266,Z 467.47,A -85,B 0,C 180,E1 -11988.351,E2 -11988.351} C_VEL
LIN {X 0,Y 389.986,Z 455.179,A -85,B 0,C 180,E1 -11988.86,E2 -11988.86} C_VEL
LIN {X 0,Y 390.414,Z 442.294,A -85,B 0,C 180,E1 -11989.196,E2 -11989.196} C_VEL
LIN {X 0,Y 391.419,Z 371.218,A -85,B 0,C 180,E1 -11990.526,E2 -11990.526} C_VEL
LIN {X 0,Y 387.148,Z 346.619,A -85,B 0,C 180,E1 -11991.289,E2 -11991.289} C_VEL
LIN {X 0,Y 385.765,Z 339.875,A -85,B 0,C 180,E1 -11991.541,E2 -11991.541} C_VEL
LIN {X 0,Y 387.203,Z 324.434,A -85,B 0,C 180,E1 -11994.833,E2 -11994.833} C_VEL
LIN {X 0,Y 387.079,Z 321.27,A -85,B 0,C 180,E1 -11995.545,E2 -11995.545} C_VEL
LIN {X 0,Y 384.692,Z 309.657,A -85,B 0,C 180,E1 -11998.359,E2 -11998.359} C_VEL
LIN {X 0,Y 383.005,Z 302.779,A -85,B 0,C 180,E1 -12000.113,E2 -12000.113} C_VEL
LIN {X 0,Y 383.005,Z 302.773,A -85,B 0,C 180,E1 -12003.401,E2 -12003.401} C_VEL
LIN {X 0,Y 383.034,Z 302.776,A -85,B 0,C 180,E1 -12006.164,E2 -12006.164} C_VEL
LIN {X 0,Y 383.009,Z 302.777,A -85,B 0,C 180,E1 -12009.958,E2 -12009.958} C_VEL
LIN {X 0,Y 383.007,Z 302.777,A -85,B 0,C 180,E1 -12012.778,E2 -12012.778} C_VEL
LIN {X 0,Y 382.998,Z 302.776,A -85,B 0,C 180,E1 -12015.789,E2 -12015.789} C_VEL
LIN {X 0,Y 382.989,Z 302.779,A -85,B 0,C 180,E1 -12018.796,E2 -12018.796} C_VEL
LIN {X 0,Y 382.999,Z 302.774,A -85,B 0,C 180,E1 -12022.096,E2 -12022.096} C_VEL
LIN {X 0,Y 383.018,Z 302.769,A -85,B 0,C 180,E1 -12025.332,E2 -12025.332} C_VEL
LIN {X 0,Y 382.983,Z 302.776,A -85,B 0,C 180,E1 -12029.081,E2 -12029.081} C_VEL
LIN {X 0,Y 383.057,Z 302.768,A -85,B 0,C 180,E1 -12032.698,E2 -12032.698} C_VEL
LIN {X 0,Y 383.033,Z 302.768,A -85,B 0,C 180,E1 -12036.192,E2 -12036.192} C_VEL
LIN {X 0,Y 383.055,Z 302.769,A -85,B 0,C 180,E1 -12039.598,E2 -12039.598} C_VEL
LIN {X 0,Y 383.104,Z 302.76,A -85,B 0,C 180,E1 -12042.931,E2 -12042.931} C_VEL
LIN {X 0,Y 383.125,Z 302.754,A -85,B 0,C 180,E1 -12046.464,E2 -12046.464} C_VEL
LIN {X 0,Y 383.15,Z 302.749,A -85,B 0,C 180,E1 -12050.498,E2 -12050.498} C_VEL
LIN {X 0,Y 383.282,Z 302.736,A -85,B 0,C 180,E1 -12053.683,E2 -12053.683} C_VEL
LIN {X 0,Y 383.384,Z 302.723,A -85,B 0,C 180,E1 -12057.899,E2 -12057.899} C_VEL
LIN {X 0,Y 383.516,Z 302.706,A -85,B 0,C 180,E1 -12060,E2 -12060} C_VEL
LIN {X 0,Y 383.245,Z 302.734,A -85,B 0,C 180,E1 -12063.154,E2 -12063.154} C_VEL
LIN {X 0,Y 383.266,Z 302.737,A -85,B 0,C 180,E1 -12066.633,E2 -12066.633} C_VEL
LIN {X 0,Y 383.259,Z 302.739,A -85,B 0,C 180,E1 -12068.436,E2 -12068.436} C_VEL
LIN {X 0,Y 383.096,Z 302.759,A -85,B 0,C 180,E1 -12071.642,E2 -12071.642} C_VEL
LIN {X 0,Y 383.109,Z 302.761,A -85,B 0,C 180,E1 -12074.882,E2 -12074.882} C_VEL
LIN {X 0,Y 383.088,Z 302.764,A -85,B 0,C 180,E1 -12078.172,E2 -12078.172} C_VEL
LIN {X 0,Y 382.991,Z 302.773,A -85,B 0,C 180,E1 -12081.531,E2 -12081.531} C_VEL
LIN {X 0,Y 383.05,Z 302.767,A -85,B 0,C 180,E1 -12084.96,E2 -12084.96} C_VEL
LIN {X 0,Y 383.029,Z 302.766,A -85,B 0,C 180,E1 -12088.27,E2 -12088.27} C_VEL
LIN {X 0,Y 383.008,Z 302.768,A -85,B 0,C 180,E1 -12092.15,E2 -12092.15} C_VEL
LIN {X 0,Y 383.017,Z 302.771,A -85,B 0,C 180,E1 -12094.668,E2 -12094.668} C_VEL
LIN {X 0,Y 382.998,Z 302.774,A -85,B 0,C 180,E1 -12097.903,E2 -12097.903} C_VEL
LIN {X 0,Y 382.984,Z 302.781,A -85,B 0,C 180,E1 -12101.347,E2 -12101.347} C_VEL
LIN {X 0,Y 382.995,Z 302.775,A -85,B 0,C 180,E1 -12104.303,E2 -12104.303} C_VEL
LIN {X 0,Y 383.01,Z 302.775,A -85,B 0,C 180,E1 -12107.24,E2 -12107.24} C_VEL
LIN {X 0,Y 383.013,Z 302.776,A -85,B 0,C 180,E1 -12110.414,E2 -12110.414} C_VEL
LIN {X 0,Y 383.025,Z 302.773,A -85,B 0,C 180,E1 -12114.044,E2 -12114.044} C_VEL
LIN {X 0,Y 383.08,Z 302.888,A -85,B 0,C 180,E1 -12115.601,E2 -12115.601} C_VEL
LIN {X 0,Y 385.587,Z 314.274,A -85,B 0,C 180,E1 -12118.514,E2 -12118.514} C_VEL
LIN {X 0,Y 388.65,Z 322.772,A -85,B 0,C 180,E1 -12118.893,E2 -12118.893} C_VEL
LIN {X 0,Y 392.034,Z 337.47,A -85,B 0,C 180,E1 -12119.407,E2 -12119.407} C_VEL
LIN {X 0,Y 390.463,Z 421.885,A -85,B 0,C 180,E1 -12120.997,E2 -12120.997} C_VEL
LIN {X 0,Y 389.858,Z 435.302,A -85,B 0,C 180,E1 -12121.463,E2 -12121.463} C_VEL
LIN {X 0,Y 389.304,Z 447.735,A -85,B 0,C 180,E1 -12122.12,E2 -12122.12} C_VEL
LIN {X 0,Y 388.409,Z 459.977,A -85,B 0,C 180,E1 -12122.994,E2 -12122.994} C_VEL
LIN {X 0,Y 387.386,Z 471.351,A -85,B 0,C 180,E1 -12124.044,E2 -12124.044} C_VEL
LIN {X 0,Y 386.336,Z 481.867,A -85,B 0,C 180,E1 -12125.266,E2 -12125.266} C_VEL
LIN {X 0,Y 385.272,Z 491.225,A -85,B 0,C 180,E1 -12126.624,E2 -12126.624} C_VEL
LIN {X 0,Y 384.24,Z 500.285,A -85,B 0,C 180,E1 -12128.26,E2 -12128.26} C_VEL
LIN {X 0,Y 383.432,Z 507.471,A -85,B 0,C 180,E1 -12129.899,E2 -12129.899} C_VEL
LIN {X 0,Y 382.662,Z 513.97,A -85,B 0,C 180,E1 -12131.806,E2 -12131.806} C_VEL
LIN {X 0,Y 382.242,Z 518.203,A -85,B 0,C 180,E1 -12133.442,E2 -12133.442} C_VEL
LIN {X 0,Y 381.884,Z 521.325,A -85,B 0,C 180,E1 -12135.069,E2 -12135.069} C_VEL
LIN {X 0,Y 381.738,Z 522.859,A -85,B 0,C 180,E1 -12136.152,E2 -12136.152} C_VEL
LIN {X 0,Y 381.694,Z 524.034,A -85,B 0,C 180,E1 -12137.388,E2 -12137.388} C_VEL
LIN {X 0,Y 381.52,Z 524.852,A -85,B 0,C 180,E1 -12139.384,E2 -12139.384} C_VEL
LIN {X 0,Y 381.504,Z 524.718,A -85,B 0,C 180,E1 -12140.456,E2 -12140.456} C_VEL
LIN {X 0,Y 381.564,Z 524.146,A -85,B 0,C 180,E1 -12141.526,E2 -12141.526} C_VEL
LIN {X 0,Y 381.769,Z 521.83,A -85,B 0,C 180,E1 -12143.658,E2 -12143.658} C_VEL
LIN {X 0,Y 381.85,Z 518.982,A -85,B 0,C 180,E1 -12145.249,E2 -12145.249} C_VEL
LIN {X 0,Y 382.107,Z 515.109,A -85,B 0,C 180,E1 -12146.836,E2 -12146.836} C_VEL
LIN {X 0,Y 382.363,Z 510.124,A -85,B 0,C 180,E1 -12148.42,E2 -12148.42} C_VEL
LIN {X 0,Y 382.865,Z 503.855,A -85,B 0,C 180,E1 -12149.999,E2 -12149.999} C_VEL
LIN {X 0,Y 383.557,Z 496.007,A -85,B 0,C 180,E1 -12151.574,E2 -12151.574} C_VEL
LIN {X 0,Y 384.169,Z 488.033,A -85,B 0,C 180,E1 -12152.883,E2 -12152.883} C_VEL
LIN {X 0,Y 384.912,Z 478.317,A -85,B 0,C 180,E1 -12154.188,E2 -12154.188} C_VEL
LIN {X 0,Y 385.825,Z 467.448,A -85,B 0,C 180,E1 -12155.356,E2 -12155.356} C_VEL
LIN {X 0,Y 386.682,Z 456.786,A -85,B 0,C 180,E1 -12156.26,E2 -12156.26} C_VEL
LIN {X 0,Y 387.327,Z 444.037,A -85,B 0,C 180,E1 -12157.1,E2 -12157.1} C_VEL
LIN {X 0,Y 387.591,Z 435.575,A -85,B 0,C 180,E1 -12157.528,E2 -12157.528} C_VEL
LIN {X 0,Y 387.01,Z 429.939,A -85,B 0,C 180,E1 -12157.789,E2 -12157.789} C_VEL
LIN {X 0,Y 384.577,Z 420.699,A -85,B 0,C 180,E1 -12158.189,E2 -12158.189} C_VEL
LIN {X 0,Y 382.114,Z 411.344,A -85,B 0,C 180,E1 -12158.495,E2 -12158.495} C_VEL
LIN {X 0,Y 381.592,Z 405.538,A -85,B 0,C 180,E1 -12158.626,E2 -12158.626} C_VEL
LIN {X 0,Y 382.483,Z 337.257,A -85,B 0,C 180,E1 -12159.903,E2 -12159.903} C_VEL
LIN {X 0,Y 378.459,Z 315.868,A -85,B 0,C 180,E1 -12160.51,E2 -12160.51} C_VEL
LIN {X 0,Y 377.957,Z 313.942,A -85,B 0,C 180,E1 -12160.588,E2 -12160.588} C_VEL
LIN {X 0,Y 376.126,Z 303.634,A -85,B 0,C 180,E1 -12163.212,E2 -12163.212} C_VEL
LIN {X 0,Y 376.022,Z 303.648,A -85,B 0,C 180,E1 -12166.281,E2 -12166.281} C_VEL
LIN {X 0,Y 375.994,Z 303.646,A -85,B 0,C 180,E1 -12169.66,E2 -12169.66} C_VEL
LIN {X 0,Y 375.971,Z 303.648,A -85,B 0,C 180,E1 -12173.659,E2 -12173.659} C_VEL
LIN {X 0,Y 375.91,Z 303.663,A -85,B 0,C 180,E1 -12176.659,E2 -12176.659} C_VEL
LIN {X 0,Y 375.91,Z 303.658,A -85,B 0,C 180,E1 -12179.083,E2 -12179.083} C_VEL
LIN {X 0,Y 375.953,Z 303.651,A -85,B 0,C 180,E1 -12181.561,E2 -12181.561} C_VEL
LIN {X 0,Y 375.953,Z 303.652,A -85,B 0,C 180,E1 -12185.415,E2 -12185.415} C_VEL
LIN {X 0,Y 375.932,Z 303.654,A -85,B 0,C 180,E1 -12188.262,E2 -12188.262} C_VEL
LIN {X 0,Y 375.912,Z 303.657,A -85,B 0,C 180,E1 -12191.597,E2 -12191.597} C_VEL
LIN {X 0,Y 375.92,Z 303.657,A -85,B 0,C 180,E1 -12194.73,E2 -12194.73} C_VEL
LIN {X 0,Y 375.925,Z 303.654,A -85,B 0,C 180,E1 -12198.399,E2 -12198.399} C_VEL
LIN {X 0,Y 375.941,Z 303.652,A -85,B 0,C 180,E1 -12200.535,E2 -12200.535} C_VEL
LIN {X 0,Y 375.956,Z 303.655,A -85,B 0,C 180,E1 -12203.495,E2 -12203.495} C_VEL
LIN {X 0,Y 375.953,Z 303.652,A -85,B 0,C 180,E1 -12205.888,E2 -12205.888} C_VEL
LIN {X 0,Y 375.957,Z 303.655,A -85,B 0,C 180,E1 -12209.687,E2 -12209.687} C_VEL
LIN {X 0,Y 375.988,Z 303.647,A -85,B 0,C 180,E1 -12212.141,E2 -12212.141} C_VEL
LIN {X 0,Y 375.996,Z 303.645,A -85,B 0,C 180,E1 -12214.538,E2 -12214.538} C_VEL
LIN {X 0,Y 375.948,Z 303.654,A -85,B 0,C 180,E1 -12218.045,E2 -12218.045} C_VEL
LIN {X 0,Y 376.016,Z 303.646,A -85,B 0,C 180,E1 -12221.474,E2 -12221.474} C_VEL
LIN {X 0,Y 376.053,Z 303.638,A -85,B 0,C 180,E1 -12224.832,E2 -12224.832} C_VEL
LIN {X 0,Y 376.042,Z 303.645,A -85,B 0,C 180,E1 -12228.136,E2 -12228.136} C_VEL
LIN {X 0,Y 376.184,Z 303.627,A -85,B 0,C 180,E1 -12231.947,E2 -12231.947} C_VEL
LIN {X 0,Y 376.155,Z 303.627,A -85,B 0,C 180,E1 -12234.64,E2 -12234.64} C_VEL
LIN {X 0,Y 376.343,Z 303.604,A -85,B 0,C 180,E1 -12237.86,E2 -12237.86} C_VEL
LIN {X 0,Y 376.478,Z 303.588,A -85,B 0,C 180,E1 -12240,E2 -12240} C_VEL
LIN {X 0,Y 376.177,Z 303.623,A -85,B 0,C 180,E1 -12243.213,E2 -12243.213} C_VEL
LIN {X 0,Y 376.233,Z 303.622,A -85,B 0,C 180,E1 -12246.435,E2 -12246.435} C_VEL
LIN {X 0,Y 376.112,Z 303.631,A -85,B 0,C 180,E1 -12249.682,E2 -12249.682} C_VEL
LIN {X 0,Y 376.082,Z 303.634,A -85,B 0,C 180,E1 -12253.658,E2 -12253.658} C_VEL
LIN {X 0,Y 376.036,Z 303.64,A -85,B 0,C 180,E1 -12257.607,E2 -12257.607} C_VEL
LIN {X 0,Y 375.971,Z 303.655,A -85,B 0,C 180,E1 -12260.833,E2 -12260.833} C_VEL
LIN {X 0,Y 375.987,Z 303.647,A -85,B 0,C 180,E1 -12264.282,E2 -12264.282} C_VEL
LIN {X 0,Y 376.013,Z 303.646,A -85,B 0,C 180,E1 -12266.653,E2 -12266.653} C_VEL
LIN {X 0,Y 375.971,Z 303.655,A -85,B 0,C 180,E1 -12269.079,E2 -12269.079} C_VEL
LIN {X 0,Y 375.951,Z 303.654,A -85,B 0,C 180,E1 -12272.829,E2 -12272.829} C_VEL
LIN {X 0,Y 375.953,Z 303.656,A -85,B 0,C 180,E1 -12275.416,E2 -12275.416} C_VEL
LIN {X 0,Y 375.971,Z 303.648,A -85,B 0,C 180,E1 -12278.272,E2 -12278.272} C_VEL
LIN {X 0,Y 375.931,Z 303.658,A -85,B 0,C 180,E1 -12281.602,E2 -12281.602} C_VEL
LIN {X 0,Y 375.924,Z 303.658,A -85,B 0,C 180,E1 -12285.269,E2 -12285.269} C_VEL
LIN {X 0,Y 375.93,Z 303.653,A -85,B 0,C 180,E1 -12288.4,E2 -12288.4} C_VEL
LIN {X 0,Y 375.969,Z 303.655,A -85,B 0,C 180,E1 -12291.731,E2 -12291.731} C_VEL
LIN {X 0,Y 375.978,Z 303.649,A -85,B 0,C 180,E1 -12295.334,E2 -12295.334} C_VEL
LIN {X 0,Y 375.956,Z 303.651,A -85,B 0,C 180,E1 -12298.439,E2 -12298.439} C_VEL
LIN {X 0,Y 376.065,Z 303.695,A -85,B 0,C 180,E1 -12301.355,E2 -12301.355} C_VEL
LIN {X 0,Y 378.624,Z 316.87,A -85,B 0,C 180,E1 -12304.434,E2 -12304.434} C_VEL
LIN {X 0,Y 379.163,Z 320.537,A -85,B 0,C 180,E1 -12305.264,E2 -12305.264} C_VEL
LIN {X 0,Y 377.878,Z 337.25,A -85,B 0,C 180,E1 -12308.815,E2 -12308.815} C_VEL
LIN {X 0,Y 377.655,Z 340.081,A -85,B 0,C 180,E1 -12309.412,E2 -12309.412} C_VEL
LIN {X 0,Y 382.168,Z 373.372,A -85,B 0,C 180,E1 -12310.284,E2 -12310.284} C_VEL
LIN {X 0,Y 381.093,Z 449.236,A -85,B 0,C 180,E1 -12311.73,E2 -12311.73} C_VEL
LIN {X 0,Y 380.453,Z 463.12,A -85,B 0,C 180,E1 -12312.22,E2 -12312.22} C_VEL
LIN {X 0,Y 379.764,Z 476.087,A -85,B 0,C 180,E1 -12312.916,E2 -12312.916} C_VEL
LIN {X 0,Y 378.806,Z 488.689,A -85,B 0,C 180,E1 -12313.842,E2 -12313.842} C_VEL
LIN {X 0,Y 377.93,Z 499.934,A -85,B 0,C 180,E1 -12314.91,E2 -12314.91} C_VEL
LIN {X 0,Y 377.26,Z 509.034,A -85,B 0,C 180,E1 -12315.986,E2 -12315.986} C_VEL
LIN {X 0,Y 376.478,Z 518.351,A -85,B 0,C 180,E1 -12317.33,E2 -12317.33} C_VEL
LIN {X 0,Y 375.671,Z 527.392,A -85,B 0,C 180,E1 -12318.945,E2 -12318.945} C_VEL
LIN {X 0,Y 375.143,Z 534.669,A -85,B 0,C 180,E1 -12320.566,E2 -12320.566} C_VEL
LIN {X 0,Y 374.851,Z 539.573,A -85,B 0,C 180,E1 -12321.917,E2 -12321.917} C_VEL
LIN {X 0,Y 374.623,Z 544.331,A -85,B 0,C 180,E1 -12323.538,E2 -12323.538} C_VEL
LIN {X 0,Y 374.554,Z 547.961,A -85,B 0,C 180,E1 -12325.157,E2 -12325.157} C_VEL
LIN {X 0,Y 374.486,Z 550.561,A -85,B 0,C 180,E1 -12326.773,E2 -12326.773} C_VEL
LIN {X 0,Y 374.524,Z 551.785,A -85,B 0,C 180,E1 -12327.85,E2 -12327.85} C_VEL
LIN {X 0,Y 374.586,Z 552.572,A -85,B 0,C 180,E1 -12328.926,E2 -12328.926} C_VEL
LIN {X 0,Y 374.589,Z 552.945,A -85,B 0,C 180,E1 -12330.001,E2 -12330.001} C_VEL
LIN {X 0,Y 374.555,Z 552.93,A -85,B 0,C 180,E1 -12331.076,E2 -12331.076} C_VEL
LIN {X 0,Y 374.497,Z 552.528,A -85,B 0,C 180,E1 -12332.152,E2 -12332.152} C_VEL
LIN {X 0,Y 374.463,Z 551.714,A -85,B 0,C 180,E1 -12333.228,E2 -12333.228} C_VEL
LIN {X 0,Y 374.552,Z 550.478,A -85,B 0,C 180,E1 -12334.305,E2 -12334.305} C_VEL
LIN {X 0,Y 374.587,Z 547.567,A -85,B 0,C 180,E1 -12336.072,E2 -12336.072} C_VEL
LIN {X 0,Y 374.892,Z 542.81,A -85,B 0,C 180,E1 -12338.083,E2 -12338.083} C_VEL
LIN {X 0,Y 375.44,Z 536.727,A -85,B 0,C 180,E1 -12339.972,E2 -12339.972} C_VEL
LIN {X 0,Y 376.11,Z 530.092,A -85,B 0,C 180,E1 -12341.589,E2 -12341.589} C_VEL
LIN {X 0,Y 377.184,Z 521.878,A -85,B 0,C 180,E1 -12343.195,E2 -12343.195} C_VEL
LIN {X 0,Y 378.104,Z 513.292,A -85,B 0,C 180,E1 -12344.564,E2 -12344.564} C_VEL
LIN {X 0,Y 379.167,Z 503.187,A -85,B 0,C 180,E1 -12345.867,E2 -12345.867} C_VEL
LIN {X 0,Y 380.433,Z 491.594,A -85,B 0,C 180,E1 -12347.054,E2 -12347.054} C_VEL
LIN {X 0,Y 381.622,Z 480.132,A -85,B 0,C 180,E1 -12347.967,E2 -12347.967} C_VEL
LIN {X 0,Y 382.577,Z 468.282,A -85,B 0,C 180,E1 -12348.683,E2 -12348.683} C_VEL
LIN {X 0,Y 383.381,Z 455.527,A -85,B 0,C 180,E1 -12349.232,E2 -12349.232} C_VEL
LIN {X 0,Y 383.837,Z 442.828,A -85,B 0,C 180,E1 -12349.579,E2 -12349.579} C_VEL
LIN {X 0,Y 384.914,Z 372.343,A -85,B 0,C 180,E1 -12350.921,E2 -12350.921} C_VEL
LIN {X 0,Y 381.105,Z 349.857,A -85,B 0,C 180,E1 -12351.63,E2 -12351.63} C_VEL
LIN {X 0,Y 378.967,Z 339.702,A -85,B 0,C 180,E1 -12351.988,E2 -12351.988} C_VEL
LIN {X 0,Y 380.358,Z 325.167,A -85,B 0,C 180,E1 -12355.15,E2 -12355.15} C_VEL
LIN {X 0,Y 379.682,Z 320.005,A -85,B 0,C 180,E1 -12356.375,E2 -12356.375} C_VEL
LIN {X 0,Y 377.143,Z 308.406,A -85,B 0,C 180,E1 -12359.286,E2 -12359.286} C_VEL
LIN {X 0,Y 375.963,Z 303.654,A -85,B 0,C 180,E1 -12360.557,E2 -12360.557} C_VEL
LIN {X 0,Y 375.962,Z 303.656,A -85,B 0,C 180,E1 -12364.111,E2 -12364.111} C_VEL
LIN {X 0,Y 375.955,Z 303.655,A -85,B 0,C 180,E1 -12366.741,E2 -12366.741} C_VEL
LIN {X 0,Y 375.989,Z 303.651,A -85,B 0,C 180,E1 -12369.97,E2 -12369.97} C_VEL
LIN {X 0,Y 375.931,Z 303.657,A -85,B 0,C 180,E1 -12373.766,E2 -12373.766} C_VEL
LIN {X 0,Y 375.935,Z 303.655,A -85,B 0,C 180,E1 -12376.81,E2 -12376.81} C_VEL
LIN {X 0,Y 375.962,Z 303.651,A -85,B 0,C 180,E1 -12380.537,E2 -12380.537} C_VEL
LIN {X 0,Y 375.964,Z 303.65,A -85,B 0,C 180,E1 -12383.495,E2 -12383.495} C_VEL
LIN {X 0,Y 375.96,Z 303.646,A -85,B 0,C 180,E1 -12385.888,E2 -12385.888} C_VEL
LIN {X 0,Y 375.965,Z 303.648,A -85,B 0,C 180,E1 -12389.687,E2 -12389.687} C_VEL
LIN {X 0,Y 376.02,Z 303.643,A -85,B 0,C 180,E1 -12393.348,E2 -12393.348} C_VEL
LIN {X 0,Y 375.996,Z 303.646,A -85,B 0,C 180,E1 -12396.888,E2 -12396.888} C_VEL
LIN {X 0,Y 375.997,Z 303.644,A -85,B 0,C 180,E1 -12400.339,E2 -12400.339} C_VEL
LIN {X 0,Y 376.029,Z 303.644,A -85,B 0,C 180,E1 -12403.719,E2 -12403.719} C_VEL
LIN {X 0,Y 376.103,Z 303.63,A -85,B 0,C 180,E1 -12407.042,E2 -12407.042} C_VEL
LIN {X 0,Y 376.118,Z 303.625,A -85,B 0,C 180,E1 -12410.318,E2 -12410.318} C_VEL
LIN {X 0,Y 376.24,Z 303.614,A -85,B 0,C 180,E1 -12413.565,E2 -12413.565} C_VEL
LIN {X 0,Y 376.35,Z 303.599,A -85,B 0,C 180,E1 -12417.859,E2 -12417.859} C_VEL
LIN {X 0,Y 376.486,Z 303.581,A -85,B 0,C 180,E1 -12420,E2 -12420} C_VEL
LIN {X 0,Y 376.183,Z 303.614,A -85,B 0,C 180,E1 -12423.213,E2 -12423.213} C_VEL
LIN {X 0,Y 376.231,Z 303.613,A -85,B 0,C 180,E1 -12426.625,E2 -12426.625} C_VEL
LIN {X 0,Y 376.204,Z 303.619,A -85,B 0,C 180,E1 -12428.595,E2 -12428.595} C_VEL
LIN {X 0,Y 376.048,Z 303.638,A -85,B 0,C 180,E1 -12431.863,E2 -12431.863} C_VEL
LIN {X 0,Y 376.057,Z 303.638,A -85,B 0,C 180,E1 -12435.167,E2 -12435.167} C_VEL
LIN {X 0,Y 376.023,Z 303.648,A -85,B 0,C 180,E1 -12438.526,E2 -12438.526} C_VEL
LIN {X 0,Y 375.957,Z 303.65,A -85,B 0,C 180,E1 -12441.955,E2 -12441.955} C_VEL
LIN {X 0,Y 376.005,Z 303.644,A -85,B 0,C 180,E1 -12445.461,E2 -12445.461} C_VEL
LIN {X 0,Y 375.96,Z 303.651,A -85,B 0,C 180,E1 -12449.08,E2 -12449.08} C_VEL
LIN {X 0,Y 375.948,Z 303.652,A -85,B 0,C 180,E1 -12452.829,E2 -12452.829} C_VEL
LIN {X 0,Y 375.957,Z 303.653,A -85,B 0,C 180,E1 -12455.416,E2 -12455.416} C_VEL
LIN {X 0,Y 375.972,Z 303.648,A -85,B 0,C 180,E1 -12458.27,E2 -12458.27} C_VEL
LIN {X 0,Y 375.934,Z 303.658,A -85,B 0,C 180,E1 -12461.601,E2 -12461.601} C_VEL
LIN {X 0,Y 375.927,Z 303.658,A -85,B 0,C 180,E1 -12465.269,E2 -12465.269} C_VEL
LIN {X 0,Y 375.934,Z 303.654,A -85,B 0,C 180,E1 -12468.399,E2 -12468.399} C_VEL
LIN {X 0,Y 375.972,Z 303.649,A -85,B 0,C 180,E1 -12471.73,E2 -12471.73} C_VEL
LIN {X 0,Y 376.016,Z 303.661,A -85,B 0,C 180,E1 -12475.16,E2 -12475.16} C_VEL
LIN {X 0,Y 378.47,Z 314.539,A -85,B 0,C 180,E1 -12478.019,E2 -12478.019} C_VEL
LIN {X 0,Y 382.44,Z 325.147,A -85,B 0,C 180,E1 -12478.517,E2 -12478.517} C_VEL
LIN {X 0,Y 385.573,Z 339.271,A -85,B 0,C 180,E1 -12479.016,E2 -12479.016} C_VEL
LIN {X 0,Y 383.895,Z 422.275,A -85,B 0,C 180,E1 -12480.603,E2 -12480.603} C_VEL
LIN {X 0,Y 383.268,Z 435.652,A -85,B 0,C 180,E1 -12481.076,E2 -12481.076} C_VEL
LIN {X 0,Y 382.653,Z 448.519,A -85,B 0,C 180,E1 -12481.772,E2 -12481.772} C_VEL
LIN {X 0,Y 381.778,Z 459.885,A -85,B 0,C 180,E1 -12482.599,E2 -12482.599} C_VEL
LIN {X 0,Y 380.672,Z 471.637,A -85,B 0,C 180,E1 -12483.699,E2 -12483.699} C_VEL
LIN {X 0,Y 379.549,Z 482.18,A -85,B 0,C 180,E1 -12484.945,E2 -12484.945} C_VEL
LIN {X 0,Y 378.558,Z 490.661,A -85,B 0,C 180,E1 -12486.184,E2 -12486.184} C_VEL
LIN {X 0,Y 377.576,Z 498.469,A -85,B 0,C 180,E1 -12487.568,E2 -12487.568} C_VEL
LIN {X 0,Y 376.692,Z 506.073,A -85,B 0,C 180,E1 -12489.238,E2 -12489.238} C_VEL
LIN {X 0,Y 375.923,Z 512.125,A -85,B 0,C 180,E1 -12490.903,E2 -12490.903} C_VEL
LIN {X 0,Y 375.36,Z 517.246,A -85,B 0,C 180,E1 -12492.725,E2 -12492.725} C_VEL
LIN {X 0,Y 374.85,Z 521.365,A -85,B 0,C 180,E1 -12494.782,E2 -12494.782} C_VEL
LIN {X 0,Y 374.684,Z 522.948,A -85,B 0,C 180,E1 -12495.886,E2 -12495.886} C_VEL
LIN {X 0,Y 374.605,Z 524.32,A -85,B 0,C 180,E1 -12497.311,E2 -12497.311} C_VEL
LIN {X 0,Y 374.441,Z 525.098,A -85,B 0,C 180,E1 -12499.181,E2 -12499.181} C_VEL
LIN {X 0,Y 374.403,Z 525.02,A -85,B 0,C 180,E1 -12500.273,E2 -12500.273} C_VEL
LIN {X 0,Y 374.46,Z 524.513,A -85,B 0,C 180,E1 -12501.364,E2 -12501.364} C_VEL
LIN {X 0,Y 374.555,Z 523.591,A -85,B 0,C 180,E1 -12502.452,E2 -12502.452} C_VEL
LIN {X 0,Y 374.697,Z 521.96,A -85,B 0,C 180,E1 -12503.77,E2 -12503.77} C_VEL
LIN {X 0,Y 374.769,Z 518.377,A -85,B 0,C 180,E1 -12505.698,E2 -12505.698} C_VEL
LIN {X 0,Y 375.088,Z 514.231,A -85,B 0,C 180,E1 -12507.315,E2 -12507.315} C_VEL
LIN {X 0,Y 375.494,Z 507.928,A -85,B 0,C 180,E1 -12509.195,E2 -12509.195} C_VEL
LIN {X 0,Y 376.149,Z 501.057,A -85,B 0,C 180,E1 -12510.802,E2 -12510.802} C_VEL
LIN {X 0,Y 376.862,Z 492.469,A -85,B 0,C 180,E1 -12512.404,E2 -12512.404} C_VEL
LIN {X 0,Y 377.526,Z 483.691,A -85,B 0,C 180,E1 -12513.735,E2 -12513.735} C_VEL
LIN {X 0,Y 378.35,Z 474.038,A -85,B 0,C 180,E1 -12514.928,E2 -12514.928} C_VEL
LIN {X 0,Y 379.285,Z 464.838,A -85,B 0,C 180,E1 -12515.849,E2 -12515.849} C_VEL
LIN {X 0,Y 379.994,Z 453.548,A -85,B 0,C 180,E1 -12516.771,E2 -12516.771} C_VEL
LIN {X 0,Y 380.583,Z 441.948,A -85,B 0,C 180,E1 -12517.493,E2 -12517.493} C_VEL
LIN {X 0,Y 380.877,Z 429.611,A -85,B 0,C 180,E1 -12518.054,E2 -12518.054} C_VEL
LIN {X 0,Y 381.379,Z 418.382,A -85,B 0,C 180,E1 -12518.377,E2 -12518.377} C_VEL
LIN {X 0,Y 381.592,Z 405.538,A -85,B 0,C 180,E1 -12518.626,E2 -12518.626} C_VEL
LIN {X 0,Y 381.056,Z 399.725,A -85,B 0,C 180,E1 -12518.761,E2 -12518.761} C_VEL
LIN {X 0,Y 375.833,Z 380.993,A -85,B 0,C 180,E1 -12519.355,E2 -12519.355} C_VEL
LIN {X 0,Y 375.248,Z 375.181,A -85,B 0,C 180,E1 -12519.496,E2 -12519.496} C_VEL
LIN {X 0,Y 375.713,Z 338.251,A -85,B 0,C 180,E1 -12520.202,E2 -12520.202} C_VEL
LIN {X 0,Y 371.713,Z 317.22,A -85,B 0,C 180,E1 -12520.815,E2 -12520.815} C_VEL
LIN {X 0,Y 370.848,Z 314.246,A -85,B 0,C 180,E1 -12520.924,E2 -12520.924} C_VEL
LIN {X 0,Y 369.066,Z 304.512,A -85,B 0,C 180,E1 -12523.447,E2 -12523.447} C_VEL
LIN {X 0,Y 368.966,Z 304.525,A -85,B 0,C 180,E1 -12526.601,E2 -12526.601} C_VEL
LIN {X 0,Y 368.934,Z 304.527,A -85,B 0,C 180,E1 -12530.052,E2 -12530.052} C_VEL
LIN {X 0,Y 368.916,Z 304.528,A -85,B 0,C 180,E1 -12533.877,E2 -12533.877} C_VEL
LIN {X 0,Y 368.855,Z 304.536,A -85,B 0,C 180,E1 -12537.211,E2 -12537.211} C_VEL
LIN {X 0,Y 368.89,Z 304.53,A -85,B 0,C 180,E1 -12539.691,E2 -12539.691} C_VEL
LIN {X 0,Y 368.893,Z 304.534,A -85,B 0,C 180,E1 -12543.042,E2 -12543.042} C_VEL
LIN {X 0,Y 368.912,Z 304.528,A -85,B 0,C 180,E1 -12546.196,E2 -12546.196} C_VEL
LIN {X 0,Y 368.87,Z 304.54,A -85,B 0,C 180,E1 -12548.956,E2 -12548.956} C_VEL
LIN {X 0,Y 368.865,Z 304.533,A -85,B 0,C 180,E1 -12552.007,E2 -12552.007} C_VEL
LIN {X 0,Y 368.873,Z 304.539,A -85,B 0,C 180,E1 -12555.175,E2 -12555.175} C_VEL
LIN {X 0,Y 368.874,Z 304.532,A -85,B 0,C 180,E1 -12558.176,E2 -12558.176} C_VEL
LIN {X 0,Y 368.875,Z 304.538,A -85,B 0,C 180,E1 -12561.364,E2 -12561.364} C_VEL
LIN {X 0,Y 368.93,Z 304.53,A -85,B 0,C 180,E1 -12565.146,E2 -12565.146} C_VEL
LIN {X 0,Y 368.922,Z 304.528,A -85,B 0,C 180,E1 -12569.046,E2 -12569.046} C_VEL
LIN {X 0,Y 368.972,Z 304.527,A -85,B 0,C 180,E1 -12571.563,E2 -12571.563} C_VEL
LIN {X 0,Y 368.991,Z 304.52,A -85,B 0,C 180,E1 -12574.019,E2 -12574.019} C_VEL
LIN {X 0,Y 368.914,Z 304.533,A -85,B 0,C 180,E1 -12577.604,E2 -12577.604} C_VEL
LIN {X 0,Y 368.975,Z 304.52,A -85,B 0,C 180,E1 -12581.107,E2 -12581.107} C_VEL
LIN {X 0,Y 368.992,Z 304.518,A -85,B 0,C 180,E1 -12584.535,E2 -12584.535} C_VEL
LIN {X 0,Y 368.997,Z 304.523,A -85,B 0,C 180,E1 -12587.907,E2 -12587.907} C_VEL
LIN {X 0,Y 369.084,Z 304.506,A -85,B 0,C 180,E1 -12591.238,E2 -12591.238} C_VEL
LIN {X 0,Y 369.127,Z 304.504,A -85,B 0,C 180,E1 -12594.537,E2 -12594.537} C_VEL
LIN {X 0,Y 369.309,Z 304.48,A -85,B 0,C 180,E1 -12597.819,E2 -12597.819} C_VEL
LIN {X 0,Y 369.448,Z 304.464,A -85,B 0,C 180,E1 -12600,E2 -12600} C_VEL
LIN {X 0,Y 369.308,Z 304.483,A -85,B 0,C 180,E1 -12602.181,E2 -12602.181} C_VEL
LIN {X 0,Y 369.193,Z 304.499,A -85,B 0,C 180,E1 -12606.559,E2 -12606.559} C_VEL
LIN {X 0,Y 369.113,Z 304.507,A -85,B 0,C 180,E1 -12608.762,E2 -12608.762} C_VEL
LIN {X 0,Y 368.998,Z 304.518,A -85,B 0,C 180,E1 -12612.094,E2 -12612.094} C_VEL
LIN {X 0,Y 368.99,Z 304.518,A -85,B 0,C 180,E1 -12615.465,E2 -12615.465} C_VEL
LIN {X 0,Y 368.951,Z 304.529,A -85,B 0,C 180,E1 -12618.895,E2 -12618.895} C_VEL
LIN {X 0,Y 368.925,Z 304.528,A -85,B 0,C 180,E1 -12622.396,E2 -12622.396} C_VEL
LIN {X 0,Y 368.993,Z 304.517,A -85,B 0,C 180,E1 -12625.981,E2 -12625.981} C_VEL
LIN {X 0,Y 368.962,Z 304.525,A -85,B 0,C 180,E1 -12628.814,E2 -12628.814} C_VEL
LIN {X 0,Y 368.904,Z 304.528,A -85,B 0,C 180,E1 -12632.238,E2 -12632.238} C_VEL
LIN {X 0,Y 368.924,Z 304.53,A -85,B 0,C 180,E1 -12635.002,E2 -12635.002} C_VEL
LIN {X 0,Y 368.905,Z 304.529,A -85,B 0,C 180,E1 -12638.642,E2 -12638.642} C_VEL
LIN {X 0,Y 368.878,Z 304.533,A -85,B 0,C 180,E1 -12642.011,E2 -12642.011} C_VEL
LIN {X 0,Y 368.877,Z 304.535,A -85,B 0,C 180,E1 -12645.177,E2 -12645.177} C_VEL
LIN {X 0,Y 368.879,Z 304.533,A -85,B 0,C 180,E1 -12648.179,E2 -12648.179} C_VEL
LIN {X 0,Y 368.904,Z 304.532,A -85,B 0,C 180,E1 -12651.361,E2 -12651.361} C_VEL
LIN {X 0,Y 368.934,Z 304.526,A -85,B 0,C 180,E1 -12655.148,E2 -12655.148} C_VEL
LIN {X 0,Y 368.928,Z 304.526,A -85,B 0,C 180,E1 -12659.048,E2 -12659.048} C_VEL
LIN {X 0,Y 368.985,Z 304.586,A -85,B 0,C 180,E1 -12661.101,E2 -12661.101} C_VEL
LIN {X 0,Y 371.276,Z 316.251,A -85,B 0,C 180,E1 -12663.89,E2 -12663.89} C_VEL
LIN {X 0,Y 372.17,Z 321.078,A -85,B 0,C 180,E1 -12665.016,E2 -12665.016} C_VEL
LIN {X 0,Y 371.097,Z 335.403,A -85,B 0,C 180,E1 -12668.123,E2 -12668.123} C_VEL
LIN {X 0,Y 370.754,Z 339.899,A -85,B 0,C 180,E1 -12669.091,E2 -12669.091} C_VEL
LIN {X 0,Y 375.375,Z 373.813,A -85,B 0,C 180,E1 -12669.986,E2 -12669.986} C_VEL
LIN {X 0,Y 374.3,Z 448.203,A -85,B 0,C 180,E1 -12671.422,E2 -12671.422} C_VEL
LIN {X 0,Y 373.682,Z 461.583,A -85,B 0,C 180,E1 -12671.887,E2 -12671.887} C_VEL
LIN {X 0,Y 372.981,Z 473.835,A -85,B 0,C 180,E1 -12672.525,E2 -12672.525} C_VEL
LIN {X 0,Y 372.085,Z 486.175,A -85,B 0,C 180,E1 -12673.401,E2 -12673.401} C_VEL
LIN {X 0,Y 371.157,Z 497.838,A -85,B 0,C 180,E1 -12674.488,E2 -12674.488} C_VEL
LIN {X 0,Y 370.323,Z 508.339,A -85,B 0,C 180,E1 -12675.718,E2 -12675.718} C_VEL
LIN {X 0,Y 369.491,Z 517.754,A -85,B 0,C 180,E1 -12677.086,E2 -12677.086} C_VEL
LIN {X 0,Y 368.665,Z 526.852,A -85,B 0,C 180,E1 -12678.733,E2 -12678.733} C_VEL
LIN {X 0,Y 368.104,Z 534.179,A -85,B 0,C 180,E1 -12680.384,E2 -12680.384} C_VEL
LIN {X 0,Y 367.787,Z 539.125,A -85,B 0,C 180,E1 -12681.761,E2 -12681.761} C_VEL
LIN {X 0,Y 367.554,Z 543.923,A -85,B 0,C 180,E1 -12683.413,E2 -12683.413} C_VEL
LIN {X 0,Y 367.473,Z 547.589,A -85,B 0,C 180,E1 -12685.063,E2 -12685.063} C_VEL
LIN {X 0,Y 367.402,Z 550.223,A -85,B 0,C 180,E1 -12686.711,E2 -12686.711} C_VEL
LIN {X 0,Y 367.425,Z 551.463,A -85,B 0,C 180,E1 -12687.808,E2 -12687.808} C_VEL
LIN {X 0,Y 367.487,Z 552.283,A -85,B 0,C 180,E1 -12688.905,E2 -12688.905} C_VEL
LIN {X 0,Y 367.505,Z 552.673,A -85,B 0,C 180,E1 -12690.001,E2 -12690.001} C_VEL
LIN {X 0,Y 367.457,Z 552.672,A -85,B 0,C 180,E1 -12691.096,E2 -12691.096} C_VEL
LIN {X 0,Y 367.396,Z 552.287,A -85,B 0,C 180,E1 -12692.193,E2 -12692.193} C_VEL
LIN {X 0,Y 367.381,Z 551.503,A -85,B 0,C 180,E1 -12693.291,E2 -12693.291} C_VEL
LIN {X 0,Y 367.457,Z 550.284,A -85,B 0,C 180,E1 -12694.388,E2 -12694.388} C_VEL
LIN {X 0,Y 367.514,Z 547.652,A -85,B 0,C 180,E1 -12696.064,E2 -12696.064} C_VEL
LIN {X 0,Y 367.721,Z 544.121,A -85,B 0,C 180,E1 -12697.689,E2 -12697.689} C_VEL
LIN {X 0,Y 368.143,Z 539.449,A -85,B 0,C 180,E1 -12699.339,E2 -12699.339} C_VEL
LIN {X 0,Y 368.886,Z 532.433,A -85,B 0,C 180,E1 -12701.262,E2 -12701.262} C_VEL
LIN {X 0,Y 369.885,Z 524.862,A -85,B 0,C 180,E1 -12702.901,E2 -12702.901} C_VEL
LIN {X 0,Y 371.001,Z 515.963,A -85,B 0,C 180,E1 -12704.446,E2 -12704.446} C_VEL
LIN {X 0,Y 371.859,Z 507.759,A -85,B 0,C 180,E1 -12705.624,E2 -12705.624} C_VEL
LIN {X 0,Y 373.105,Z 497.364,A -85,B 0,C 180,E1 -12706.835,E2 -12706.835} C_VEL
LIN {X 0,Y 374.178,Z 487.412,A -85,B 0,C 180,E1 -12707.771,E2 -12707.771} C_VEL
LIN {X 0,Y 375.415,Z 474.775,A -85,B 0,C 180,E1 -12708.699,E2 -12708.699} C_VEL
LIN {X 0,Y 376.38,Z 461.67,A -85,B 0,C 180,E1 -12709.392,E2 -12709.392} C_VEL
LIN {X 0,Y 377.105,Z 448.746,A -85,B 0,C 180,E1 -12709.848,E2 -12709.848} C_VEL
LIN {X 0,Y 378.545,Z 374.179,A -85,B 0,C 180,E1 -12711.308,E2 -12711.308} C_VEL
LIN {X 0,Y 374.71,Z 351.275,A -85,B 0,C 180,E1 -12712.046,E2 -12712.046} C_VEL
LIN {X 0,Y 372.246,Z 339.276,A -85,B 0,C 180,E1 -12712.507,E2 -12712.507} C_VEL
LIN {X 0,Y 373.521,Z 326.137,A -85,B 0,C 180,E1 -12715.425,E2 -12715.425} C_VEL
LIN {X 0,Y 371.848,Z 316.917,A -85,B 0,C 180,E1 -12717.714,E2 -12717.714} C_VEL
LIN {X 0,Y 369.223,Z 305.887,A -85,B 0,C 180,E1 -12720.609,E2 -12720.609} C_VEL
LIN {X 0,Y 368.912,Z 304.533,A -85,B 0,C 180,E1 -12720.987,E2 -12720.987} C_VEL
LIN {X 0,Y 368.938,Z 304.529,A -85,B 0,C 180,E1 -12724.853,E2 -12724.853} C_VEL
LIN {X 0,Y 368.908,Z 304.533,A -85,B 0,C 180,E1 -12728.64,E2 -12728.64} C_VEL
LIN {X 0,Y 368.883,Z 304.536,A -85,B 0,C 180,E1 -12732.009,E2 -12732.009} C_VEL
LIN {X 0,Y 368.881,Z 304.535,A -85,B 0,C 180,E1 -12735.176,E2 -12735.176} C_VEL
LIN {X 0,Y 368.884,Z 304.533,A -85,B 0,C 180,E1 -12738.177,E2 -12738.177} C_VEL
LIN {X 0,Y 368.908,Z 304.53,A -85,B 0,C 180,E1 -12741.36,E2 -12741.36} C_VEL
LIN {X 0,Y 368.937,Z 304.525,A -85,B 0,C 180,E1 -12745.146,E2 -12745.146} C_VEL
LIN {X 0,Y 368.93,Z 304.526,A -85,B 0,C 180,E1 -12749.046,E2 -12749.046} C_VEL
LIN {X 0,Y 368.976,Z 304.522,A -85,B 0,C 180,E1 -12751.563,E2 -12751.563} C_VEL
LIN {X 0,Y 369,Z 304.517,A -85,B 0,C 180,E1 -12754.02,E2 -12754.02} C_VEL
LIN {X 0,Y 368.932,Z 304.526,A -85,B 0,C 180,E1 -12757.605,E2 -12757.605} C_VEL
LIN {X 0,Y 368.982,Z 304.518,A -85,B 0,C 180,E1 -12761.107,E2 -12761.107} C_VEL
LIN {X 0,Y 368.997,Z 304.515,A -85,B 0,C 180,E1 -12764.535,E2 -12764.535} C_VEL
LIN {X 0,Y 369.004,Z 304.517,A -85,B 0,C 180,E1 -12767.907,E2 -12767.907} C_VEL
LIN {X 0,Y 369.166,Z 304.499,A -85,B 0,C 180,E1 -12771.869,E2 -12771.869} C_VEL
LIN {X 0,Y 369.142,Z 304.491,A -85,B 0,C 180,E1 -12774.537,E2 -12774.537} C_VEL
LIN {X 0,Y 369.315,Z 304.476,A -85,B 0,C 180,E1 -12777.819,E2 -12777.819} C_VEL
LIN {X 0,Y 369.455,Z 304.457,A -85,B 0,C 180,E1 -12780,E2 -12780} C_VEL
LIN {X 0,Y 369.315,Z 304.475,A -85,B 0,C 180,E1 -12782.181,E2 -12782.181} C_VEL
LIN {X 0,Y 369.201,Z 304.489,A -85,B 0,C 180,E1 -12786.612,E2 -12786.612} C_VEL
LIN {X 0,Y 369.137,Z 304.5,A -85,B 0,C 180,E1 -12788.761,E2 -12788.761} C_VEL
LIN {X 0,Y 369.004,Z 304.515,A -85,B 0,C 180,E1 -12792.093,E2 -12792.093} C_VEL
LIN {X 0,Y 368.997,Z 304.516,A -85,B 0,C 180,E1 -12795.465,E2 -12795.465} C_VEL
LIN {X 0,Y 368.982,Z 304.523,A -85,B 0,C 180,E1 -12798.893,E2 -12798.893} C_VEL
LIN {X 0,Y 368.924,Z 304.529,A -85,B 0,C 180,E1 -12802.396,E2 -12802.396} C_VEL
LIN {X 0,Y 368.999,Z 304.516,A -85,B 0,C 180,E1 -12805.98,E2 -12805.98} C_VEL
LIN {X 0,Y 368.914,Z 304.527,A -85,B 0,C 180,E1 -12809.69,E2 -12809.69} C_VEL
LIN {X 0,Y 368.896,Z 304.533,A -85,B 0,C 180,E1 -12813.043,E2 -12813.043} C_VEL
LIN {X 0,Y 368.916,Z 304.528,A -85,B 0,C 180,E1 -12816.197,E2 -12816.197} C_VEL
LIN {X 0,Y 368.902,Z 304.533,A -85,B 0,C 180,E1 -12818.953,E2 -12818.953} C_VEL
LIN {X 0,Y 368.881,Z 304.533,A -85,B 0,C 180,E1 -12822.009,E2 -12822.009} C_VEL
LIN {X 0,Y 368.879,Z 304.535,A -85,B 0,C 180,E1 -12825.176,E2 -12825.176} C_VEL
LIN {X 0,Y 368.882,Z 304.534,A -85,B 0,C 180,E1 -12828.177,E2 -12828.177} C_VEL
LIN {X 0,Y 368.907,Z 304.532,A -85,B 0,C 180,E1 -12831.36,E2 -12831.36} C_VEL
LIN {X 0,Y 368.955,Z 304.692,A -85,B 0,C 180,E1 -12834.77,E2 -12834.77} C_VEL
LIN {X 0,Y 371.179,Z 314.558,A -85,B 0,C 180,E1 -12837.474,E2 -12837.474} C_VEL
LIN {X 0,Y 376.202,Z 327.192,A -85,B 0,C 180,E1 -12838.117,E2 -12838.117} C_VEL
LIN {X 0,Y 379.092,Z 339.979,A -85,B 0,C 180,E1 -12838.587,E2 -12838.587} C_VEL
LIN {X 0,Y 377.356,Z 422.672,A -85,B 0,C 180,E1 -12840.196,E2 -12840.196} C_VEL
LIN {X 0,Y 376.697,Z 436.002,A -85,B 0,C 180,E1 -12840.676,E2 -12840.676} C_VEL
LIN {X 0,Y 376.026,Z 449.007,A -85,B 0,C 180,E1 -12841.394,E2 -12841.394} C_VEL
LIN {X 0,Y 375.134,Z 460.194,A -85,B 0,C 180,E1 -12842.223,E2 -12842.223} C_VEL
LIN {X 0,Y 373.98,Z 471.939,A -85,B 0,C 180,E1 -12843.341,E2 -12843.341} C_VEL
LIN {X 0,Y 372.88,Z 481.708,A -85,B 0,C 180,E1 -12844.507,E2 -12844.507} C_VEL
LIN {X 0,Y 371.856,Z 490.087,A -85,B 0,C 180,E1 -12845.728,E2 -12845.728} C_VEL
LIN {X 0,Y 370.811,Z 498.059,A -85,B 0,C 180,E1 -12847.136,E2 -12847.136} C_VEL
LIN {X 0,Y 369.841,Z 505.782,A -85,B 0,C 180,E1 -12848.835,E2 -12848.835} C_VEL
LIN {X 0,Y 369.007,Z 511.937,A -85,B 0,C 180,E1 -12850.53,E2 -12850.53} C_VEL
LIN {X 0,Y 368.406,Z 516.768,A -85,B 0,C 180,E1 -12852.228,E2 -12852.228} C_VEL
LIN {X 0,Y 367.994,Z 520.43,A -85,B 0,C 180,E1 -12853.923,E2 -12853.923} C_VEL
LIN {X 0,Y 367.629,Z 523.032,A -85,B 0,C 180,E1 -12855.61,E2 -12855.61} C_VEL
LIN {X 0,Y 367.524,Z 524.603,A -85,B 0,C 180,E1 -12857.226,E2 -12857.226} C_VEL
LIN {X 0,Y 367.374,Z 525.344,A -85,B 0,C 180,E1 -12858.971,E2 -12858.971} C_VEL
LIN {X 0,Y 367.371,Z 524.872,A -85,B 0,C 180,E1 -12861.196,E2 -12861.196} C_VEL
LIN {X 0,Y 367.443,Z 523.998,A -85,B 0,C 180,E1 -12862.305,E2 -12862.305} C_VEL
LIN {X 0,Y 367.615,Z 522.224,A -85,B 0,C 180,E1 -12863.786,E2 -12863.786} C_VEL
LIN {X 0,Y 367.691,Z 518.949,A -85,B 0,C 180,E1 -12865.615,E2 -12865.615} C_VEL
LIN {X 0,Y 367.998,Z 514.896,A -85,B 0,C 180,E1 -12867.263,E2 -12867.263} C_VEL
LIN {X 0,Y 368.392,Z 508.693,A -85,B 0,C 180,E1 -12869.18,E2 -12869.18} C_VEL
LIN {X 0,Y 369.07,Z 501.929,A -85,B 0,C 180,E1 -12870.818,E2 -12870.818} C_VEL
LIN {X 0,Y 369.811,Z 493.53,A -85,B 0,C 180,E1 -12872.45,E2 -12872.45} C_VEL
LIN {X 0,Y 370.495,Z 484.905,A -85,B 0,C 180,E1 -12873.806,E2 -12873.806} C_VEL
LIN {X 0,Y 371.423,Z 474.278,A -85,B 0,C 180,E1 -12875.156,E2 -12875.156} C_VEL
LIN {X 0,Y 372.39,Z 465.069,A -85,B 0,C 180,E1 -12876.093,E2 -12876.093} C_VEL
LIN {X 0,Y 373.123,Z 453.767,A -85,B 0,C 180,E1 -12877.032,E2 -12877.032} C_VEL
LIN {X 0,Y 373.727,Z 442.144,A -85,B 0,C 180,E1 -12877.767,E2 -12877.767} C_VEL
